(* POU FB_KL3208Config, ST *)
FUNCTION_BLOCK FB_KL3208Config
VAR_INPUT
	bConfigurate		: BOOL; 		(*Rising edge starts configuration including read-configuration afterwards*)
	bReadConfig			: BOOL;			(*Rising edge reads the actual configuration*)
	iSetSensorType		: INT;			(*Sensor-type to be set, see table*)
	tTimeout			: TIME :=t#5s;	(*Time-out-time for Reading/Configuration - initially set to 5s*)
END_VAR
VAR_OUTPUT
	bBusy				: BOOL;			(*Reading or configuration is in progress*)
	bError				: BOOL;			(*Error while reading/configuration*)
	iErrorId			: UDINT;		(*Id of the last upcoming error*)
	iState				: USINT;		(*As long as the funcion-block is not busy, this variable shows the state of the terminal, otherwise it is 0*)
	iDataIn				: INT;			(*As long as the funcion-block is not busy, this variable shows the dataIn of the terminal, otherwise it keeps the value previous to reding/configuration*)
	iTerminalType		: WORD;			(*Terminal-type-number, in this case 3208*)
	iSpecialType		: WORD;			(*Sub-type-number*)
	iFirmwareVersion	: WORD;			(*Firmware in ASCII-code*)
	sDescription		: STRING;		(*Terminal-type, special-type and firmware-version as readable text*)
	sSensorType			: STRING;		(*Text-description of entered sensor-type*)
END_VAR
VAR
	rtRead				: R_TRIG;
	rtSet				: R_TRIG;
	bSetReq				: BOOL;
	tonTimeout			: TON;
	iStep				: INT;
	bSetConfigError		: BOOL;
	wReg32				: WORD;
	wSetReg32			: WORD;
	wReg39				: WORD;
	wSetReg39			: WORD;
	wFirmware			: WORD;
	pFirmware			: POINTER TO WORD;
	sFirmware			: STRING(2);
	iDataInSaved		: INT;
END_VAR
VAR_IN_OUT
	stInData   			: ST_KL3208InData;	(* Process image of the inputs. *)
	stOutData 			: ST_KL3208OutData;	(* Process image of the outputs. *)
END_VAR
tonTimeout	(PT:=tTimeout);
IF	tonTimeout.Q	THEN
	bError			:= TRUE;
	iErrorId		:= 16#8001;
	iStep			:= 0;
END_IF

rtSet	(CLK:=bConfigurate);
rtRead	(CLK:=bReadConfig);

IF	(rtSet.Q OR rtRead.Q)	AND NOT bBusy THEN
	bBusy			:= TRUE;
	bError			:= FALSE;
	iErrorId		:= 0;
	iDataInSaved	:= stInData.iDataIn;
	tonTimeout.IN	:= TRUE;
	iStep			:= 10;
	IF	rtSet.Q	THEN
		bSetReq	:= TRUE;
	END_IF
END_IF

IF bBusy THEN
	iDataIn		:= iDataInSaved;
	iState		:= 0;
ELSE
	iDataIn		:= stInData.iDataIn;
	iState		:= stInData.iState;
END_IF


CASE iStep OF

0:	(*idle*)
	bBusy				:= FALSE;
	bSetReq				:= FALSE;
	tonTimeout.IN		:= FALSE;

10:	(*Klemmentyp (Kl32xx) auslesen: Register 8*)
	stOutData.iCtrl	:= 16#88;	(*Register 8 Lesen*)

	IF stInData.iState = 16#88 THEN
		iTerminalType	:= INT_TO_WORD(stInData.iDataIn);
		iStep:=20;
	END_IF

20:	(*Spezialtyp (Kl32xx-yyy) auslesen: Register 29*)
	stOutData.iCtrl	:= 16#9D;	(*Register 29 Lesen*)

	IF stInData.iState = 16#9D THEN
		iSpecialType	:= INT_TO_WORD(stInData.iDataIn);
		iStep:=30;
	END_IF

30:	(*Firmware auslesen: Register 9*)
	stOutData.iCtrl	:= 16#89;	(*Register 9 Lesen*)

	IF stInData.iState = 16#89 THEN
		iFirmwareVersion:= INT_TO_WORD(stInData.iDataIn);
		(*Umwandlung in STRING*)
		wFirmware		:= iFirmwareVersion;
		wFirmware		:= ROR(wFirmware,8);(*Reihenfolge der beiden Zeichen der Firmware tauschen*)
		pFirmware		:= ADR(sFirmware);	(*Einen Pointer auf den Info-String (Ausgang) legen*)
		pFirmware^		:= wFirmware;		(*Diesen Adressbereich mit dem richtig getauschen Wert beschreiben - damit ist auch der String beschrieben*)

		sDescription	:= CONCAT('Terminal ',WORD_TO_STRING(iTerminalType));

		CASE LEN(WORD_TO_STRING(iSpecialType)) OF
			1: sDescription	:= CONCAT(sDescription,'-000');
			2: sDescription	:= CONCAT(sDescription,'-00');
			3: sDescription	:= CONCAT(sDescription,'-0');
		ELSE
			sDescription	:= CONCAT(sDescription,'-');
		END_CASE

		sDescription	:= CONCAT(sDescription,WORD_TO_STRING(iSpecialType));
		sDescription	:= CONCAT(sDescription,' / Firmware ');
		sDescription	:= CONCAT(sDescription,sFirmware);

		IF bSetReq	THEN
			iStep:=100;
		ELSE
			iStep:=150;
		END_IF
	END_IF

	(*Falscher Klemmentyp angeschlossen, Konfiguration vorzeitig abbrechen*)
	IF (iTerminalType <> 3208)	THEN
		bError		:= TRUE;
		iErrorId	:= 16#8002;
		iStep		:= 160;
	END_IF

(*-----------------------------------------------------------------*)

100:(*jetzige Sensoreinstellung lesen: Register 32*)
	stOutData.iCtrl	:= 16#A0;	(*Register 32 Lesen*)

	IF stInData.iState = 16#A0 THEN
		wReg32			:= INT_TO_WORD(stInData.iDataIn);
		iStep:=105;
	END_IF

105:(*jetzige Sensoreinstellung lesen: Register 39*)
	stOutData.iCtrl	:= 16#A7;	(*Register 39 Lesen*)

	IF stInData.iState = 16#A7 THEN
		wReg39			:= INT_TO_WORD(stInData.iDataIn);
		A_SetConfigTable;			(*entsprechende Einstellungen vornehmen*)
		iStep:=110;
		IF	bSetConfigError	THEN
			iStep:=150;
		END_IF
	END_IF

110:(*Codewort Register 31 setzen: 16#1235 -> Schreibschutz aufheben*)
	stOutData.iCtrl	:= 16#DF;	(*Register 31 beschreiben*)
	stOutData.iDataOut	:= 16#1235;	(*Nutzdaten: Codewort*)

	IF stInData.iState = 16#9F THEN
		stOutData.iCtrl	:= 16#9F;	(*Register 31 Auslesen*)
		iStep:=120;
	END_IF

120:(*Bestätigung Codewort gesetzt erfragen*)
	IF	stInData.iDataIn	= 16#1235	THEN
		iStep:=130;
	END_IF

130:(*Nun Register 32 mit dem neuen Wert beschreiben*)
	stOutData.iCtrl	:= 16#E0;	(*Register 32 beschreiben*)
	stOutData.iDataOut	:= WORD_TO_INT(wSetReg32);

	IF stInData.iState = 16#A0 THEN
		iStep:=135;
	END_IF

135:(*Und Register 39 mit dem neuen Wert beschreiben*)
	stOutData.iCtrl	:= 16#E7;	(*Register 39 beschreiben*)
	stOutData.iDataOut	:= WORD_TO_INT(wSetReg39);

	IF stInData.iState = 16#A7 THEN
		iStep:=140;
	END_IF

140:(*Codewort Register 31 löschen: 16#0000 -> Schreibschutz setzen*)
	stOutData.iCtrl	:= 16#DF;	(*Register 31 beschreiben*)
	stOutData.iDataOut	:= 16#0000;

	IF stInData.iState = 16#9F THEN
		iStep:=150;
	END_IF

150:(*nach erfolgter Parametrierung Sensoreinstellung lesen: Register 32*)
	stOutData.iCtrl	:= 16#A0;	(*Register 32 Lesen*)

	IF stInData.iState = 16#A0 THEN
		wReg32			:= INT_TO_WORD(stInData.iDataIn);
		iStep:=155;
	END_IF

155:(*nach erfolgter Parametrierung Sensoreinstellung lesen: Register 39*)
	stOutData.iCtrl	:= 16#A7;	(*Register 39 Lesen*)

	IF stInData.iState = 16#A7 THEN
		wReg39			:= INT_TO_WORD(stInData.iDataIn);
		A_ReadConfigTable;
		iStep:=160;
	END_IF

160:(*Registerkommunikation beenden*)
	stOutData.iCtrl	:= 0; (*auch alle anderen Steuerbits mit ablöschen*)
	(*Rückmeldeabfrage Prozessdatenaustausch (Bit7) noch aktiv? *)
	(*alle anderen Bits könnten durch einen bestimmten Signalpegel gesetzt sein *)
	IF stInData.iState.7 = FALSE THEN
		iStep:=0;
	END_IF

END_CASE
END_FUNCTION_BLOCK
ACTION A_ReadConfigTable:
(*IF Reg39 is set to 0, Reg32 is responsible for the sensor-type, otherwise Reg39 sets the sensor*)

IF	wReg39=0	THEN
	CASE (SHR(wReg32,12)) OF	(*Check sensor-type via the 4 most significant bits*)
		2#0000: sSensorType	:= 'PT1000';
		2#0001: sSensorType	:= 'NI1000';
		2#0010: sSensorType	:= 'RSNI1000';
	ELSE
		sSensorType	:='Unknown';
		bError		:= TRUE;
		iErrorId	:= 16#8021;
	END_CASE
ELSE
	CASE wReg39 OF
		16#32: sSensorType	:= 'NCT1K8';
		16#33: sSensorType	:= 'NCT1K8_TK';
		16#34: sSensorType	:= 'NCT2K2';
		16#35: sSensorType	:= 'NCT3K';
		16#36: sSensorType	:= 'NCT5K';
		16#37: sSensorType	:= 'NTC10K';
		16#38: sSensorType	:= 'NTC10KPRE';
		16#39: sSensorType	:= 'NTC10K_3204';
		16#3A: sSensorType	:= 'NTC10KTYP2';
		16#3B: sSensorType	:= 'NTC10KTYP3';
		16#3C: sSensorType	:= 'NTC10KDALE';
		16#3D: sSensorType	:= 'NTC10K3A221';
		16#3E: sSensorType	:= 'NTC20K';
		16#64: sSensorType	:= 'Poti, Resolution 0,1 Ohm';
		16#65: sSensorType	:= 'Poti, Resolution 1 Ohm';
		16#C8: sSensorType	:= 'NTC100K';
		16#FF: sSensorType	:= 'User defined';
	ELSE
		sSensorType	:='Unknown';
		bError		:= TRUE;
		iErrorId	:= 16#8021;
	END_CASE
END_IF
END_ACTION
ACTION A_SetConfigTable:
bSetConfigError	:= FALSE;

CASE iSetSensorType OF	(*Then set the sensor-type via the 4 most significant bits*)

	0:	wSetReg32	:= wReg32		AND 2#0000111111111111;(*First clear the first 4 bits*)
		wSetReg32	:= wSetReg32	OR 2#0000000000000000;(*PT1000*)	(*Then set the sensor-type via the 4 most significant bits*)
		wSetReg39	:= 0;

	1:	wSetReg32	:= wReg32		AND 2#0000111111111111;(*First clear the first 4 bits*)
		wSetReg32	:= wSetReg32	OR 2#0001000000000000;(*NI1000*)	(*Then set the sensor-type via the 4 most significant bits*)
		wSetReg39	:= 0;

	2:	wSetReg32	:= wReg32		AND 2#0000111111111111;(*First clear the first 4 bits*)
		wSetReg32	:= wSetReg32	OR 2#0010000000000000;(*RSNI1000*)	(*Then set the sensor-type via the 4 most significant bits*)
		wSetReg39	:= 0;


	3:	wSetReg39	:= 16#32;		(*NCT1K8*)
	4:	wSetReg39	:= 16#33;		(*NCT1K8_TK*)
	5:	wSetReg39	:= 16#34;		(*NCT2K2*)
	6:	wSetReg39	:= 16#35;		(*NCT3K*)
	7:	wSetReg39	:= 16#36;		(*NCT5K*)
	8:	wSetReg39	:= 16#37;		(*NTC10K*)
	9:	wSetReg39	:= 16#38;		(*NTC10KPRE*)
	10:	wSetReg39	:= 16#39;		(*NTC10K_3204*)
	11:	wSetReg39	:= 16#3A;		(*NTC10KTYP2*)
	12:	wSetReg39	:= 16#3B;		(*NTC10KTYP3*)
	13:	wSetReg39	:= 16#3C;		(*NTC10KDALE*)
	14:	wSetReg39	:= 16#3D;		(*NTC10K3A221*)
	15:	wSetReg39	:= 16#3E;		(*NTC20K*)
	16:	wSetReg39	:= 16#64;		(*Poti, Resolution 0,1 Ohm*)
	17:	wSetReg39	:= 16#65;		(*Poti, Resolution 1 Ohm*)
	18:	wSetReg39	:= 16#C8;		(*NTC100K*)
ELSE
	bSetConfigError	:= TRUE;
	bError			:= TRUE;
	iErrorId		:= 16#8020;
END_CASE
END_ACTION

(* POU FB_KL320xConfig, ST *)
FUNCTION_BLOCK FB_KL320xConfig
VAR_INPUT
	bConfigurate		: BOOL; 		(*Rising edge starts configuration including read-configuration afterwards*)
	bReadConfig			: BOOL;			(*Rising edge reads the actual configuration*)
	iSetSensorType		: INT;			(*Sensor-type to be set, see table*)
	tTimeout			: TIME :=t#5s;	(*Time-out-time for Reading/Configuration - initially set to 5s*)
END_VAR
VAR_OUTPUT
	bBusy				: BOOL;			(*Reading or configuration is in progress*)
	bError				: BOOL;			(*Error while reading/configuration*)
	iErrorId			: UDINT;		(*Id of the last upcoming error*)
	iState				: USINT;		(*As long as the funcion-block is not busy, this variable shows the state of the terminal, otherwise it is 0*)
	iDataIn				: INT;			(*As long as the funcion-block is not busy, this variable shows the dataIn of the terminal, otherwise it keeps the value previous to reding/configuration*)
	iTerminalType		: WORD;			(*Terminal-type-number, e.g. 3204*)
	iSpecialType		: WORD;			(*Sub-type-number*)
	iFirmwareVersion	: WORD;			(*Firmware in ASCII-code*)
	sDescription		: STRING;		(*Terminal-type, special-type and firmware-version as readable text*)
	sSensorType			: STRING;		(*Text-description of entered sensor-type*)
	bTwoWiredConnection	: BOOL;			(*Shows, if two-wired connection is selected*)
END_VAR
VAR
	rtRead				: R_TRIG;
	rtSet				: R_TRIG;
	bSetReq				: BOOL;
	tonTimeout			: TON;
	iStep				: INT;
	bSetConfigError		: BOOL;
	wReg32				: WORD;
	wSetReg32			: WORD;
	wFirmware			: WORD;
	pFirmware			: POINTER TO WORD;
	sFirmware			: STRING(2);
	iDataInSaved		: INT;
END_VAR
VAR_IN_OUT
	stInData   			: ST_KL320xInData;	(* Process image of the inputs. *)
	stOutData 			: ST_KL320xOutData;	(* Process image of the outputs. *)
END_VAR
tonTimeout	(PT:=tTimeout);
IF	tonTimeout.Q	THEN
	bError			:= TRUE;
	iErrorId		:= 16#8001;
	iStep			:= 0;
END_IF

rtSet	(CLK:=bConfigurate);
rtRead	(CLK:=bReadConfig);

IF	(rtSet.Q OR rtRead.Q)	AND NOT bBusy THEN
	bBusy			:= TRUE;
	bError			:= FALSE;
	iErrorId		:= 0;
	iDataInSaved	:= stInData.iDataIn;
	tonTimeout.IN	:= TRUE;
	iStep			:= 10;
	IF	rtSet.Q	THEN
		bSetReq	:= TRUE;
	END_IF
END_IF

IF bBusy THEN
	iDataIn		:= iDataInSaved;
	iState		:= 0;
ELSE
	iDataIn		:= stInData.iDataIn;
	iState		:= stInData.iState;
END_IF


CASE iStep OF

0:	(*idle*)
	bBusy				:= FALSE;
	bSetReq				:= FALSE;
	tonTimeout.IN		:= FALSE;

10:	(*Klemmentyp (Kl32xx) auslesen: Register 8*)
	stOutData.iCtrl	:= 16#88;	(*Register 8 Lesen*)

	IF stInData.iState = 16#88 THEN
		iTerminalType	:= INT_TO_WORD(stInData.iDataIn);
		iStep:=20;
	END_IF

20:	(*Spezialtyp (Kl32xx-yyy) auslesen: Register 29*)
	stOutData.iCtrl	:= 16#9D;	(*Register 29 Lesen*)

	IF stInData.iState = 16#9D THEN
		iSpecialType	:= INT_TO_WORD(stInData.iDataIn);
		iStep:=30;
	END_IF

30:	(*Firmware auslesen: Register 9*)
	stOutData.iCtrl	:= 16#89;	(*Register 9 Lesen*)

	IF stInData.iState = 16#89 THEN
		iFirmwareVersion:= INT_TO_WORD(stInData.iDataIn);
		(*Umwandlung in STRING*)
		wFirmware		:= iFirmwareVersion;
		wFirmware		:= ROR(wFirmware,8);(*Reihenfolge der beiden Zeichen der Firmware tauschen*)
		pFirmware		:= ADR(sFirmware);	(*Einen Pointer auf den Info-String (Ausgang) legen*)
		pFirmware^		:= wFirmware;		(*Diesen Adressbereich mit dem richtig getauschen Wert beschreiben - damit ist auch der String beschrieben*)

		sDescription	:= CONCAT('Terminal ',WORD_TO_STRING(iTerminalType));

		CASE LEN(WORD_TO_STRING(iSpecialType)) OF
			1: sDescription	:= CONCAT(sDescription,'-000');
			2: sDescription	:= CONCAT(sDescription,'-00');
			3: sDescription	:= CONCAT(sDescription,'-0');
		ELSE
			sDescription	:= CONCAT(sDescription,'-');
		END_CASE

		sDescription	:= CONCAT(sDescription,WORD_TO_STRING(iSpecialType));
		sDescription	:= CONCAT(sDescription,' / Firmware ');
		sDescription	:= CONCAT(sDescription,sFirmware);

		IF bSetReq	THEN
			iStep:=100;
		ELSE
			iStep:=150;
		END_IF
	END_IF

	(*Falscher Klemmentyp angeschlossen, Konfiguration vorzeitig abbrechen*)
	IF ((iTerminalType <> 3201)	AND (iTerminalType <> 3202) AND (iTerminalType <> 3204))	THEN
		bError		:= TRUE;
		iErrorId	:= 16#8002;
		iStep		:= 160;
	END_IF

(*-----------------------------------------------------------------*)

100:(*jetzige Sensoreinstellung lesen: Register 32*)
	stOutData.iCtrl	:= 16#A0;	(*Register 32 Lesen*)

	IF stInData.iState = 16#A0 THEN
		wReg32			:= INT_TO_WORD(stInData.iDataIn);
		A_SetConfigTable;		(*entsprechende Bits für den zu schreibenden Wert setzen, der Rest bleibt unberührt*)
		iStep:=110;
		IF	bSetConfigError	THEN
			iStep:=150;
		END_IF
	END_IF

110:(*Codewort Register 31 setzen: 16#1235 -> Schreibschutz aufheben*)
	stOutData.iCtrl	:= 16#DF;	(*Register 31 beschreiben*)
	stOutData.iDataOut	:= 16#1235;	(*Nutzdaten: Codewort*)

	IF stInData.iState = 16#9F THEN
		stOutData.iCtrl	:= 16#9F;	(*Register 31 Auslesen*)
		iStep:=120;
	END_IF

120:(*Bestätigung Codewort gesetzt erfragen*)
	IF	stInData.iDataIn	= 16#1235	THEN
		iStep:=130;
	END_IF

130:(*Nun Register 32 mit dem neuen Wert beschreiben*)
	stOutData.iCtrl	:= 16#E0;	(*Register 32 beschreiben*)
	stOutData.iDataOut	:= WORD_TO_INT(wSetReg32);

	IF stInData.iState = 16#A0 THEN
		iStep:=140;
	END_IF

140:(*Codewort Register 31 löschen: 16#0000 -> Schreibschutz setzen*)
	stOutData.iCtrl	:= 16#DF;	(*Register 31 beschreiben*)
	stOutData.iDataOut	:= 16#0000;

	IF stInData.iState = 16#9F THEN
		iStep:=150;
	END_IF

150:(*nach erfolgter Parametrierung Sensoreinstellung lesen: Register 32*)
	stOutData.iCtrl	:= 16#A0;	(*Register 32 Lesen*)

	IF stInData.iState = 16#A0 THEN
		wReg32			:= INT_TO_WORD(stInData.iDataIn);
		A_ReadConfigTable;
		iStep:=160;
	END_IF

160:(*Registerkommunikation beenden*)
	stOutData.iCtrl	:= 0; (*auch alle anderen Steuerbits mit ablöschen*)
	(*Rückmeldeabfrage Prozessdatenaustausch (Bit7) noch aktiv? *)
	(*alle anderen Bits könnten durch einen bestimmten Signalpegel gesetzt sein *)
	IF stInData.iState.7 = FALSE THEN
		iStep:=0;
	END_IF

END_CASE
END_FUNCTION_BLOCK
ACTION A_ReadConfigTable:
CASE (SHR(wReg32,12)) OF	(*Check sensor-type via the 4 most significant bits*)
	2#0000: sSensorType:='PT100';
	2#0001: sSensorType:='NI100';
	2#0010: sSensorType:='PT1000';
	2#0011: sSensorType:='PT500';
	2#0100: sSensorType:='PT200';
	2#0101: sSensorType:='NI1000';
	2#0110: sSensorType:='NI120';
	
	2#1110: sSensorType:='10Ohm .. 5000Ohm';
	2#1111: sSensorType:='10Ohm .. 1200Ohm';
ELSE
	sSensorType	:='Unknown';
	bError		:= TRUE;
	iErrorId	:= 16#802A;
END_CASE

bTwoWiredConnection:=wReg32.10;
END_ACTION
ACTION A_SetConfigTable:
bSetConfigError	:= FALSE;

wSetReg32:=wReg32 AND 2#0000111111111111;(*First clear the first 4 bits*)

CASE iSetSensorType OF	(*Then set the sensor-type via the 4 most significant bits - Bit 10 sets 2-wired-connection*)

	0:	wSetReg32:=wSetReg32 OR 2#0000000000000000;(*PT100*)
		wSetReg32.10:=FALSE;					(*1-Wired*)

	1:	wSetReg32:=wSetReg32 OR 2#0001000000000000;(*NI100*)
		wSetReg32.10:=FALSE;					(*1-Wired*)

	2:	wSetReg32:=wSetReg32 OR 2#0010000000000000;(*PT1000*)
		wSetReg32.10:=FALSE;					(*1-Wired*)

	3:	wSetReg32:=wSetReg32 OR 2#0011000000000000;(*PT500*)
		wSetReg32.10:=FALSE;					(*1-Wired*)

	4:	wSetReg32:=wSetReg32 OR 2#0100000000000000;(*PT200*)
		wSetReg32.10:=FALSE;					(*1-Wired*)

	5:	wSetReg32:=wSetReg32 OR 2#0101000000000000;(*NI1000*)
		wSetReg32.10:=FALSE;					(*1-Wired*)

	6:	wSetReg32:=wSetReg32 OR 2#0110000000000000;(*NI120*)
		wSetReg32.10:=FALSE;					(*1-Wired*)

	7:	wSetReg32:=wSetReg32 OR 2#1110000000000000;(*10Ohm .. 5000Ohm*)
		wSetReg32.10:=FALSE;					(*1-Wired*)

	8:	wSetReg32:=wSetReg32 OR 2#1111000000000000;(*10Ohm .. 1200Ohm*)
		wSetReg32.10:=FALSE;					(*1-Wired*)

	9:	wSetReg32:=wSetReg32 OR 2#0010000000000000;(*PT1000*)
		wSetReg32.10:=TRUE;						(*2-Wired*)

		IF (iTerminalType=3204)	THEN			(*2-Wired is not allowed for KL3204*)
			bSetConfigError	:= TRUE;
			bError			:= TRUE;
			iErrorId		:= 16#8028;
		END_IF
ELSE
	bSetConfigError	:= TRUE;
	bError			:= TRUE;
	iErrorId		:= 16#8029;
END_CASE
END_ACTION

(* POU FB_KL3228Config, ST *)
FUNCTION_BLOCK FB_KL3228Config
VAR_INPUT
	bConfigurate		: BOOL; 		(*Rising edge starts configuration including read-configuration afterwards*)
	bReadConfig			: BOOL;			(*Rising edge reads the actual configuration*)
	iSetSensorType		: INT;			(*Sensor-type to be set, see table*)
	tTimeout			: TIME :=t#5s;	(*Time-out-time for Reading/Configuration - initially set to 5s*)
END_VAR
VAR_OUTPUT
	bBusy				: BOOL;			(*Reading or configuration is in progress*)
	bError				: BOOL;			(*Error while reading/configuration*)
	iErrorId			: UDINT;		(*Id of the last upcoming error*)
	iState				: USINT;		(*As long as the funcion-block is not busy, this variable shows the state of the terminal, otherwise it is 0*)
	iDataIn				: INT;			(*As long as the funcion-block is not busy, this variable shows the dataIn of the terminal, otherwise it keeps the value previous to reding/configuration*)
	iTerminalType		: WORD;			(*Terminal-type-number, in this case 3228*)
	iSpecialType		: WORD;			(*Sub-type-number*)
	iFirmwareVersion	: WORD;			(*Firmware in ASCII-code*)
	sDescription		: STRING;		(*Terminal-type, special-type and firmware-version as readable text*)
	sSensorType			: STRING;		(*Text-description of entered sensor-type*)
END_VAR
VAR
	rtRead				: R_TRIG;
	rtSet				: R_TRIG;
	bSetReq				: BOOL;
	tonTimeout			: TON;
	iStep				: INT;
	bSetConfigError		: BOOL;
	wReg32				: WORD;
	wSetReg32			: WORD;
	wFirmware			: WORD;
	pFirmware			: POINTER TO WORD;
	sFirmware			: STRING(2);
	iDataInSaved		: INT;
END_VAR
VAR_IN_OUT
	stInData   			: ST_KL3228InData;	(* Process image of the inputs. *)
	stOutData 			: ST_KL3228OutData;	(* Process image of the outputs. *)
END_VAR
tonTimeout	(PT:=tTimeout);
IF	tonTimeout.Q	THEN
	bError			:= TRUE;
	iErrorId		:= 16#8001;
	iStep			:= 0;
END_IF

rtSet	(CLK:=bConfigurate);
rtRead	(CLK:=bReadConfig);

IF	(rtSet.Q OR rtRead.Q)	AND NOT bBusy THEN
	bBusy			:= TRUE;
	bError			:= FALSE;
	iErrorId		:= 0;
	iDataInSaved	:= stInData.iDataIn;
	tonTimeout.IN	:= TRUE;
	iStep			:= 10;
	IF	rtSet.Q	THEN
		bSetReq	:= TRUE;
	END_IF
END_IF

IF bBusy THEN
	iDataIn		:= iDataInSaved;
	iState		:= 0;
ELSE
	iDataIn		:= stInData.iDataIn;
	iState		:= stInData.iState;
END_IF


CASE iStep OF

0:	(*idle*)
	bBusy				:= FALSE;
	bSetReq				:= FALSE;
	tonTimeout.IN		:= FALSE;

10:	(*Klemmentyp (Kl32xx) auslesen: Register 8*)
	stOutData.iCtrl	:= 16#88;	(*Register 8 Lesen*)

	IF stInData.iState = 16#88 THEN
		iTerminalType	:= INT_TO_WORD(stInData.iDataIn);
		iStep:=20;
	END_IF

20:	(*Spezialtyp (Kl32xx-yyy) auslesen: Register 29*)
	stOutData.iCtrl	:= 16#9D;	(*Register 29 Lesen*)

	IF stInData.iState = 16#9D THEN
		iSpecialType	:= INT_TO_WORD(stInData.iDataIn);
		iStep:=30;
	END_IF

30:	(*Firmware auslesen: Register 9*)
	stOutData.iCtrl	:= 16#89;	(*Register 9 Lesen*)

	IF stInData.iState = 16#89 THEN
		iFirmwareVersion:= INT_TO_WORD(stInData.iDataIn);
		(*Umwandlung in STRING*)
		wFirmware		:= iFirmwareVersion;
		wFirmware		:= ROR(wFirmware,8);(*Reihenfolge der beiden Zeichen der Firmware tauschen*)
		pFirmware		:= ADR(sFirmware);	(*Einen Pointer auf den Info-String (Ausgang) legen*)
		pFirmware^		:= wFirmware;		(*Diesen Adressbereich mit dem richtig getauschen Wert beschreiben - damit ist auch der String beschrieben*)

		sDescription	:= CONCAT('Terminal ',WORD_TO_STRING(iTerminalType));

		CASE LEN(WORD_TO_STRING(iSpecialType)) OF
			1: sDescription	:= CONCAT(sDescription,'-000');
			2: sDescription	:= CONCAT(sDescription,'-00');
			3: sDescription	:= CONCAT(sDescription,'-0');
		ELSE
			sDescription	:= CONCAT(sDescription,'-');
		END_CASE

		sDescription	:= CONCAT(sDescription,WORD_TO_STRING(iSpecialType));
		sDescription	:= CONCAT(sDescription,' / Firmware ');
		sDescription	:= CONCAT(sDescription,sFirmware);

		IF bSetReq	THEN
			iStep:=100;
		ELSE
			iStep:=150;
		END_IF
	END_IF

	(*Falscher Klemmentyp angeschlossen, Konfiguration vorzeitig abbrechen*)
	IF (iTerminalType <> 3228)	THEN
		bError		:= TRUE;
		iErrorId	:= 16#8002;
		iStep		:= 160;
	END_IF

(*-----------------------------------------------------------------*)

100:(*jetzige Sensoreinstellung lesen: Register 32*)
	stOutData.iCtrl	:= 16#A0;	(*Register 32 Lesen*)

	IF stInData.iState = 16#A0 THEN
		wReg32			:= INT_TO_WORD(stInData.iDataIn);
		A_SetConfigTable;		(*entsprechende Bits für den zu schreibenden Wert setzen, der Rest bleibt unberührt*)
		iStep:=110;
		IF	bSetConfigError	THEN
			iStep:=150;
		END_IF
	END_IF

110:(*Codewort Register 31 setzen: 16#1235 -> Schreibschutz aufheben*)
	stOutData.iCtrl	:= 16#DF;	(*Register 31 beschreiben*)
	stOutData.iDataOut	:= 16#1235;	(*Nutzdaten: Codewort*)

	IF stInData.iState = 16#9F THEN
		stOutData.iCtrl	:= 16#9F;	(*Register 31 Auslesen*)
		iStep:=120;
	END_IF

120:(*Bestätigung Codewort gesetzt erfragen*)
	IF	stInData.iDataIn	= 16#1235	THEN
		iStep:=130;
	END_IF

130:(*Nun Register 32 mit dem neuen Wert beschreiben*)
	stOutData.iCtrl	:= 16#E0;	(*Register 32 beschreiben*)
	stOutData.iDataOut	:= WORD_TO_INT(wSetReg32);

	IF stInData.iState = 16#A0 THEN
		iStep:=140;
	END_IF

140:(*Codewort Register 31 löschen: 16#0000 -> Schreibschutz setzen*)
	stOutData.iCtrl	:= 16#DF;	(*Register 31 beschreiben*)
	stOutData.iDataOut	:= 16#0000;

	IF stInData.iState = 16#9F THEN
		iStep:=150;
	END_IF

150:(*nach erfolgter Parametrierung Sensoreinstellung lesen: Register 32*)
	stOutData.iCtrl	:= 16#A0;	(*Register 32 Lesen*)

	IF stInData.iState = 16#A0 THEN
		wReg32			:= INT_TO_WORD(stInData.iDataIn);
		A_ReadConfigTable;
		iStep:=160;
	END_IF

160:(*Registerkommunikation beenden*)
	stOutData.iCtrl	:= 0; (*auch alle anderen Steuerbits mit ablöschen*)
	(*Rückmeldeabfrage Prozessdatenaustausch (Bit7) noch aktiv? *)
	(*alle anderen Bits könnten durch einen bestimmten Signalpegel gesetzt sein *)
	IF stInData.iState.7 = FALSE THEN
		iStep:=0;
	END_IF

END_CASE
END_FUNCTION_BLOCK
ACTION A_ReadConfigTable:
CASE (SHR(wReg32,12)) OF	(*Check sensor-type via the 4 most significant bits*)
	2#0000: sSensorType	:= 'PT1000';
	2#0001: sSensorType	:= 'NI1000';
	2#0010: sSensorType	:= 'RSNI1000';
ELSE
	sSensorType	:='Unknown';
	bError		:= TRUE;
	iErrorId	:= 16#8031;
END_CASE
END_ACTION
ACTION A_SetConfigTable:
bSetConfigError	:= FALSE;

CASE iSetSensorType OF	(*Then set the sensor-type via the 4 most significant bits*)
	0:	wSetReg32	:= wReg32		AND 2#0000111111111111;(*First clear the first 4 bits*)
		wSetReg32	:= wSetReg32	OR 2#0000000000000000;(*PT1000*)	(*Then set the sensor-type via the 4 most significant bits*)

	1:	wSetReg32	:= wReg32		AND 2#0000111111111111;(*First clear the first 4 bits*)
		wSetReg32	:= wSetReg32	OR 2#0001000000000000;(*NI1000*)	(*Then set the sensor-type via the 4 most significant bits*)

	2:	wSetReg32	:= wReg32		AND 2#0000111111111111;(*First clear the first 4 bits*)
		wSetReg32	:= wSetReg32	OR 2#0010000000000000;(*RSNI1000*)(*Then set the sensor-type via the 4 most significant bits*)
ELSE
	bSetConfigError	:= TRUE;
	bError			:= TRUE;
	iErrorId		:= 16#8030;
END_CASE
END_ACTION

(* POU FB_NovRamReadWrite, ST *)
FUNCTION_BLOCK FB_NovRamReadWrite (*if the dpram must be accessed in a special manor, this function block returns error 0x701. In this case use FB_NovRamReadWriteEx instead.*)
VAR_INPUT
	nDevId 	: UDINT;		(* Device id of the FCxxxx card. Map the FC card as generic DPRAM/NOVRAM card im System Manager *)
	bRead		: BOOL;		(* Rising edge starts read data block from NovRam*)
	bWrite		: BOOL;		(* Rising edge starts write data block to NovRam*)
	cbSrcLen	: UDINT;		(* Number of data bytes to write *)
	cbDestLen: UDINT;		(* Number of data bytes to read*)
	pSrcAddr	: UDINT;		(* Address of the write data buffer *)
	pDestAddr	: UDINT;		(* Address of the read data buffer *)
	tTimeOut	: TIME := DEFAULT_ADS_TIMEOUT;		(* Max timeout for this command *)
END_VAR
VAR_OUTPUT
	bBusy		: BOOL;		(* The fb is working *)
	bError		: BOOL;		(* The fb returns an error *)
	nErrId		: UDINT;		(* Error code *)
	cbRead	: UDINT;		(* Number of succesfully read data bytes *)
	cbWrite	: UDINT;		(* Number of succesfully write data bytes *)
END_VAR
VAR
	bInit			: BOOL := FALSE;
	nInitDevId		: UDINT	:= 0;
	bWantRead		: BOOL := FALSE;
	bWantWrite		: BOOL := FALSE;

	iStep			: BYTE := 0;
	RisingRead		: R_TRIG;
	RisingWrite		: R_TRIG;
	stNovRamAddrInfo: ST_NovRamAddrInfo;
	fbAdsReadEx		: ADSREADEX;
END_VAR
RisingRead( CLK := bRead );
RisingWrite( CLK := bWrite );

CASE iStep OF
0:
	(* idle step, wait for rising edge on fb input*)
	IF RisingRead.Q OR RisingWrite.Q THEN

		bBusy 	:= TRUE;
		bError 	:= FALSE;
		nErrId 	:= 0;
		cbRead 	:= 0;
		cbWrite := 0;

		bWantRead 	:=	RisingRead.Q;	(* Save flags *)
		bWantWrite 	:= 	RisingWrite.Q;

		IF	 (nDevId > 0) AND (pSrcAddr > 0) AND (cbSrcLen > 0) AND (pDestAddr > 0) AND (cbDestLen> 0) THEN

			IF 	( NOT bInit ) OR ( bInit AND ( nDevId <> nInitDevId)) THEN

				bInit := FALSE;

				nInitDevId	:= 	nDevId;	(* Save the devid *)
				MEMSET( ADR( stNovRamAddrInfo ) , 0, SIZEOF(stNovRamAddrInfo));

				(* Get the nov ram address pointer and the novram byte size *)
				fbAdsReadEx( READ := FALSE );(*reset the fb*)
				fbAdsReadEx(
						NETID:= '',
						PORT:= AMSPORT_R0_IO,
						IDXGRP:= 16#5000+nInitDevId,
						IDXOFFS:= 16#FFFF_0200,
						LEN:= SIZEOF(stNovRamAddrInfo),
						DESTADDR:= ADR(stNovRamAddrInfo),
						READ:= TRUE,
						TMOUT:= tTimeout);

				iStep := 10;	(* wait for the ads fb *)

			ELSIF bInit THEN

				IF bWantWrite THEN(* copy size bytes to novRAM *)
					cbWrite := MEMCPY(stNovRamAddrInfo.pCardAddress, pSrcAddr, MIN(cbSrcLen,stNovRamAddrInfo.iCardMemSize ) );
				END_IF
				IF bWantRead THEN(* copy size bytes from novRAM *)
					cbRead := MEMCPY(pDestAddr, stNovRamAddrInfo.pCardAddress, MIN(cbDestLen,stNovRamAddrInfo.iCardMemSize ));
				END_IF

				bBusy := FALSE;

			END_IF

		ELSE
			bBusy := FALSE;
			bError := TRUE;
			nErrId := 1798;(* invalid parameter value(s)*)
		END_IF
	END_IF

10:
	fbAdsReadEx( READ := FALSE );
	IF NOT fbAdsReadEx.BUSY THEN

		IF NOT fbAdsReadEx.ERR THEN
			bInit := TRUE;
			bError := FALSE;
			nErrId := 0;

			IF bWantWrite THEN(* copy size bytes to novRAM *)
				cbWrite := MEMCPY(stNovRamAddrInfo.pCardAddress, pSrcAddr, MIN(cbSrcLen,stNovRamAddrInfo.iCardMemSize ) );
			END_IF
			IF bWantRead THEN(* copy size bytes from novRAM *)
				cbRead := MEMCPY(pDestAddr, stNovRamAddrInfo.pCardAddress, MIN(cbDestLen,stNovRamAddrInfo.iCardMemSize ));
			END_IF
		ELSE
			bError := fbAdsReadEx.ERR;
			nErrId := fbAdsReadEx.ERRID;
		END_IF

		bBusy := FALSE;
		iStep := 0; (*go to the idle step and wait for the next call *)

	END_IF

END_CASE;
END_FUNCTION_BLOCK

(* POU FB_NovRamReadWriteEx, ST *)
FUNCTION_BLOCK FB_NovRamReadWriteEx (*if the dpram must be accessed in a special manor, this function block returns error 0x701. In this case use FB_NovRamReadWriteEx instead.*)
VAR_INPUT
	nDevId 		:	UDINT;		(* Device id of the FCxxxx card. Map the FC card as generic DPRAM/NOVRAM card im System Manager *)
	bRead		:	BOOL;		(* Rising edge starts read data block from NovRam*)
	bWrite		:	BOOL;		(* Rising edge starts write data block to NovRam*)
	cbSrcLen	:	UDINT;		(* Number of data bytes to write *)
	cbDestLen	:	UDINT;		(* Number of data bytes to read*)
	pSrcAddr	:	UDINT;		(* Address of the write data buffer *)
	pDestAddr	:	UDINT;		(* Address of the read data buffer *)
	nReadOffs	:	UDINT;		(* Offset in the DPRAM to start reading from*)
	nWriteOffs	:	UDINT;		(* Offset in the DPRAM to start writing to*)
	tTimeOut	: 	TIME;		(* Max timeout for this command *)
END_VAR
VAR_OUTPUT
	bBusy		:	BOOL;		(* The fb is working *)
	bError		:	BOOL;		(* The fb returns an error *)
	nErrId		:	UDINT;		(* Error code *)
	cbRead		: 	UDINT;		(* Number of succesfully read data bytes *)
	cbWrite		: 	UDINT;		(* Number of succesfully write data bytes *)
END_VAR
VAR
	bInit				: BOOL := FALSE;
	nInitDevId		: UDINT	:= 0;
	bWantRead		: BOOL := FALSE;
	bWantWrite		: BOOL := FALSE;
	bCopy			: BOOL := FALSE;

	i				: UDINT:=0;
	iStep			: BYTE := 0;
	RisingRead		: R_TRIG;
	RisingWrite		: R_TRIG;

	stNovRamAddrInfo	: ST_NovRamAddrInfoEx;
	fbAdsReadEx		: ADSREADEX;

	pByte			: POINTER TO BYTE;
	pCard			: POINTER TO BYTE;
END_VAR
RisingRead( CLK := bRead );
RisingWrite( CLK := bWrite );

CASE iStep OF
0:
	(* idle step, wait for rising edge on fb input*)
	IF RisingRead.Q OR RisingWrite.Q THEN

		bBusy 	:= TRUE;
		bError 	:= FALSE;
		nErrId 	:= 0;
		cbRead 	:= 0;
		cbWrite := 0;

		bWantRead 	:=	RisingRead.Q;	(* Save flags *)
		bWantWrite 	:= 	RisingWrite.Q;

		IF	(nDevId > 0) AND (  ( bWantWrite AND ( pSrcAddr>0) AND (cbSrcLen>0) ) OR ( bWantRead AND (pDestAddr > 0) AND (cbDestLen> 0) )  ) THEN
			IF 	( NOT bInit ) OR ( bInit AND ( nDevId <> nInitDevId)) THEN
				bInit := FALSE;

				nInitDevId	:= 	nDevId;	(* Save the devid *)
				MEMSET( ADR( stNovRamAddrInfo ), 0, 10);

				(* Get the nov ram address pointer and the novram byte size *)
				fbAdsReadEx( READ := FALSE );(*reset the fb*)
				fbAdsReadEx(
						NETID:= '',
						PORT:= AMSPORT_R0_IO,
						IDXGRP:= 16#5000+nInitDevId,
						IDXOFFS:= 16#FFFF_0201,
						LEN:= 10,
						DESTADDR:= ADR(stNovRamAddrInfo),
						READ:= TRUE,
						TMOUT:= tTimeout);

				iStep := 10;	(* wait for the ads fb *)

			ELSIF bInit THEN
				bCopy := TRUE;
				bBusy := FALSE;
			END_IF
		ELSE
			bBusy := FALSE;
			bError := TRUE;
			nErrId := 1798;(* invalid parameter value(s)*)
		END_IF
	END_IF

10:
	fbAdsReadEx( READ := FALSE );
	IF NOT fbAdsReadEx.BUSY THEN
		IF NOT fbAdsReadEx.ERR THEN
			bCopy := TRUE;
		ELSE
			bError := fbAdsReadEx.ERR;
			nErrId := fbAdsReadEx.ERRID;
			bBusy := FALSE;
		END_IF
		iStep := 0; (*go to the idle step and wait for the next call *)
	END_IF

END_CASE;

IF bCopy THEN
	IF  (bWantWrite AND (nWriteOffs <= stNovRamAddrInfo.iCardMemSize-1)) OR (bWantRead AND (nReadOffs <= stNovRamAddrInfo.iCardMemSize-1)) THEN
		CASE stNovRamAddrInfo.eAccessType OF
		eIOAccess_Default:
			IF bWantWrite THEN(* copy size bytes to novRAM *)
				cbWrite := MEMCPY(stNovRamAddrInfo.pCardAddress+nWriteOffs, pSrcAddr, MIN(cbSrcLen,stNovRamAddrInfo.iCardMemSize-nWriteOffs) );
			END_IF
			IF bWantRead THEN(* copy size bytes from novRAM *)
				cbRead := MEMCPY(pDestAddr, stNovRamAddrInfo.pCardAddress+nReadOffs, MIN(cbDestLen,stNovRamAddrInfo.iCardMemSize-nReadOffs));
			END_IF
		eIOAccess_Byte:
			IF bWantWrite THEN(* copy size bytes to novRAM *)
				cbWrite:=MIN(cbSrcLen,stNovRamAddrInfo.iCardMemSize-nWriteOffs);
				pByte := pSrcAddr;
				pCard := stNovRamAddrInfo.pCardAddress + nWriteOffs;
				FOR i:=1 TO cbWrite DO
					pCard^:= pByte^;
					pCard := pCard + 1;
					pByte := pByte + 1;
				END_FOR
			END_IF
			IF bWantRead THEN(* copy size bytes from novRAM *)
				cbRead:=MIN(cbDestLen,stNovRamAddrInfo.iCardMemSize-nReadOffs);
				pByte := pDestAddr;
				pCard := stNovRamAddrInfo.pCardAddress + nReadOffs;
				FOR i:=1 TO cbRead  DO
					pByte^:=pCard^;
					pCard := pCard + 1;
					pByte := pByte + 1;
				END_FOR
			END_IF
			bInit := TRUE;
			bError := FALSE;
			nErrId := 0;
		ELSE
			bInit := FALSE;
			bError := TRUE;
			nErrId := 16#701;
		END_CASE
	ELSE
		bInit := FALSE;
		bError := TRUE;
		nErrId := 16#706;
	END_IF
	bBusy := FALSE;
	bCopy:= FALSE;
END_IF
END_FUNCTION_BLOCK

(* POU FB_ReadAdsTecSysData, ST *)
FUNCTION_BLOCK FB_ReadAdsTecSysData
VAR_INPUT
	sNetId		: T_AmsNetId;
	bEnable		: BOOL;
	tCycleTime	: TIME := T#100ms;
END_VAR
VAR_OUTPUT
	bValid		: BOOL;
	bError		: BOOL;
	nErrId		: UDINT;
	stSysData	: ST_AdsTecSysData;
END_VAR
VAR
	dwTemp		: DWORD := 0;
	ptr			: POINTER TO ARRAY[0..3] OF SINT;
	delay		: TON;
	wPort		: WORD := 16#240;
	risingEdge	: R_TRIG;
	step 		: INT := 0;
	fbAdsRdWrtEx: ADSRDWRTEX;
END_VAR
risingEdge( CLK := bEnable );
IF risingEdge.Q THEN
	MEMSET( ADR( stSysData ), 0, SIZEOF( stSysData ) );
	delay( IN := FALSE, PT := tCycleTime );
	bValid := FALSE;
	bError := FALSE;
	nErrId := 0;
	step := 1;
ELSIF (NOT bEnable) THEN
	step := 0;
	bValid := FALSE;
END_IF

CASE step OF
	0:	; (* idle step *)

	1:	(* Wait some time and repeat reading...*)
		delay( IN := TRUE );
		IF delay.Q THEN
			fbAdsRdWrtEx(  WRTRD := FALSE );
			delay( IN := FALSE );
			step := step +1;
		END_IF
	2:
(*	AMSPORT_ROUTER						: UINT := 16#0001;
	ROUTERADSGRP_ACCESS_HARDWARE	: DWORD := 16#0005;
	ROUTERADSOFFS_A_HW_READIOPORT	: DWORD := 16#0001;
*)
		fbAdsRdWrtEx(  WRTRD := FALSE );
		fbAdsRdWrtEx( 	NetId := sNetId,
						Port := 1,
						IDXGRP := 16#05,
						IDXOFFS := 16#01,
						WRITELEN := SIZEOF(wPort),
						READLEN := SIZEOF(dwTemp),
						SRCADDR := ADR( wPort ),
						DESTADDR := ADR( dwTemp ),
						WRTRD := TRUE,
						TMOUT := tCycleTime
						);

		step := step +1;
	3:
		fbAdsRdWrtEx(  WRTRD := FALSE );
		IF NOT fbAdsRdWrtEx.BUSY THEN
			IF NOT fbAdsRdWrtEx.ERR THEN
				stSysData.bShiftKey := GETBIT32( dwTemp, 0 );
				stSysData.bRMouseKey := GETBIT32( dwTemp, 1 );
				stSysData.bHotkey := GETBIT32( dwTemp, 2 );
				stSysData.bTaskChaKey := GETBIT32( dwTemp, 3 );
				stSysData.bABCKey := GETBIT32( dwTemp, 4 );
				stSysData.bRsrv1 := GETBIT32( dwTemp, 5 );
				stSysData.bRsrv2 := GETBIT32( dwTemp,6 );
				stSysData.bRsrv3 := GETBIT32( dwTemp, 7 );

				stSysData.bMainFanErr := GETBIT32( dwTemp, 8 );
				stSysData.bCPUFanErr := GETBIT32( dwTemp, 9 );
				stSysData.bTempErr := GETBIT32( dwTemp, 10 );
				stSysData.bBatteryErr := GETBIT32( dwTemp, 11 );
				stSysData.bRsrv4 := GETBIT32( dwTemp, 12 );
				stSysData.bRsrv5 := GETBIT32( dwTemp, 13 );
				stSysData.bRsrv6 := GETBIT32( dwTemp, 14 );
				stSysData.bRsrv7 := GETBIT32( dwTemp, 15 );

				ptr := ADR( dwTemp );
				stSysData.nMainNTCTemp := ptr^[ 2 ];
				stSysData.nExtNTCTemp := ptr^[ 3 ];
				bValid := TRUE;
				step := 1;
			ELSE
				bValid := FALSE;
				bError := TRUE;
				nErrid := fbAdsRdWrtEx.ERRID;
				step := 0;
			END_IF
		END_IF

			;
END_CASE
END_FUNCTION_BLOCK

(* POU FB_ReadInput_analog, ST *)
(*********************************************************************************************************

NAME..............	:	FB_ReadInput_analog
DATE...............	:	11.07.2003
AUTHOR........	:	G.Sieder (Beckhoff Industrieelektronik)

DESCRIPTION:	FB for Read analog data from one Slave

HISTORY:	
11.07.2003	gs	start coding

*********************************************************************************************************)
FUNCTION_BLOCK FB_ReadInput_analog
VAR_INPUT
	iSlaveaddress		:BYTE;
	iChannel				:BYTE;
	bCycleMode			:BOOL;		(*0: Acyclic , 1:Cyclic (permanent Read/Write) *)
	bStart				:BOOL;
END_VAR
VAR_OUTPUT
	bBusy				:BOOL;
	bErr					:BOOL;
	iErrornumber			:BYTE;
	bValid				:BOOL;
	bOverflow			:BOOL;
	iReadValue			:WORD;

END_VAR
VAR_IN_OUT
	stParameterBuffer		:ST_ParameterBuffer;
END_VAR
VAR
	fbParameterinterface	:FB_ASI_Parameterinterface;
	bHiWord				:BOOL;
	iParametervalue		:DWORD;
	iParameterReadValue	:DWORD;
	iParametergroup		:WORD;
	iErrCounter			:BYTE;
	istate				:INT;
END_VAR
	CASE istate OF

		0:	IF bstart THEN
				bBusy		:=TRUE;
				bErr			:=FALSE;
				bOverflow	:=FALSE;
				bValid		:=FALSE;
				iErrornumber	:=0;
				(*check Slavenumber*)
				IF (iSlaveaddress>64) OR (iChannel>4) THEN
					bErr			:=TRUE;
					iErrornumber	:=ERROR_ASI_SLAVEADDRESS;
					istate		:=10;
				ELSE
					istate		:=1;
				END_IF
			END_IF

		(*prepare Parameternumber*)
		1:	iParametergroup	:=(iSlaveaddress*4)+(iChannel-1);
			istate	:=2;

		(*write Readrequest*)
		2:	fbParameterinterface(iParameternumber	:=iParametergroup+16#200,
							stParameterBuffer		:=stParameterBuffer,
							bParametermode		:=FALSE,
							bCycleMode			:=bCycleMode,
							bStart				:=TRUE);
			IF (NOT fbParameterinterface.bBusy) OR bCycleMode THEN
				IF fbParameterinterface.bErr THEN
					bErr			:=TRUE;
					IF fbParameterinterface.iErrornumber =1 THEN
						iErrornumber	:=ERROR_ASI_COMM_ERROR;
					ELSE
						FOR iErrCounter:=1 TO 3 DO
							IF ((SHR(fbParameterinterface.iErrornumber,iErrCounter-1)) AND 16#2000)<>0 THEN
								iErrornumber :=iErrCounter+10;
							END_IF
						END_FOR
					END_IF
					istate	:=10;
				ELSE
					IF (fbParameterinterface.iParameterReadvalue  AND 16#0200)<>0 THEN
						bOverflow	:=TRUE;
					ELSE
						bValid		:=TRUE;
					END_IF
					iParameterReadValue	:=fbParameterinterface.iParameterReadvalue;
					istate	:=3;
				END_IF
			END_IF

		(*read Parametervalue*)
		3:	iReadValue	:=DWORD_TO_WORD(iParameterReadValue);
			IF (NOT bStart) OR (NOT bCycleMode) THEN
				fbParameterinterface(bStart			:=FALSE,
								stParameterBuffer	:=stParameterBuffer);
				IF (NOT fbParameterinterface.bBusy) THEN
					istate	:=10;
				END_IF
			ELSE
				istate	:=1;
			END_IF

			(*Quit*)
		10:	bBusy	:=FALSE;
			IF (NOT bStart) THEN
				istate	:=0;
			END_IF

	ELSE
		;
	END_CASE
END_FUNCTION_BLOCK

(* POU FB_WriteOutput_analog, ST *)
(*********************************************************************************************************

NAME..............	:	FB_WriteOutput_analog
DATE...............	:	11.07.2003
AUTHOR........	:	G.Sieder (Beckhoff Industrieelektronik)

DESCRIPTION:	FB for Write analog data to one Slave

HISTORY:	
11.07.2003	gs	start coding

*********************************************************************************************************)
FUNCTION_BLOCK FB_WriteOutput_analog
VAR_INPUT
	iSlaveaddress		:BYTE;
	iChannel				:BYTE;
	iSlavevalue			:WORD;
	bCycleMode			:BOOL;		(*0: Acyclic , 1:Cyclic (permanent Read/Write) *)
	bStart				:BOOL;
END_VAR
VAR_OUTPUT
	bBusy				:BOOL;
	bErr					:BOOL;
	iErrornumber			:BYTE;

END_VAR
VAR_IN_OUT
	stParameterBuffer		:ST_ParameterBuffer;
END_VAR
VAR
	fbParameterinterface	:FB_ASI_Parameterinterface;
	bHiWord				:BOOL;
	iParametervalue		:DWORD;
	iParameterReadValue	:DWORD;
	iParametergroup		:WORD;
	iErrCounter			:BYTE;
	istate				:INT;

	iReadValue			:WORD;
END_VAR
	CASE istate OF

		0:	IF bstart THEN
				bBusy		:=TRUE;
				bErr			:=FALSE;
				iErrornumber	:=0;
				(*check Slavenumber*)
				IF (iSlaveaddress>64) OR (iChannel>4) THEN
					bErr			:=TRUE;
					iErrornumber	:=ERROR_ASI_SLAVEADDRESS;
					istate		:=10;
				ELSE
					istate		:=1;
				END_IF
			END_IF

		(*prepare Parameternumber and -value*)
		1:	iParametergroup	:=(iSlaveaddress*4)+(iChannel-1);
			iParametervalue	:=0;
			iParametervalue	:=iSlavevalue;
			iParametervalue	:=iParametervalue+16#10000;
			istate	:=2;

		(*write Parameter*)
		2:	fbParameterinterface(iParameternumber	:=iParametergroup+16#200,
							iParametervalue		:=iParametervalue,
							stParameterBuffer		:=stParameterBuffer,
							bParametermode		:=TRUE,
							bCycleMode			:=bCycleMode,
							bStart				:=TRUE);
			IF (NOT fbParameterinterface.bBusy) OR bCycleMode THEN
				IF fbParameterinterface.bErr THEN
					bErr			:=TRUE;
					IF fbParameterinterface.iErrornumber =1 THEN
						iErrornumber	:=ERROR_ASI_COMM_ERROR;
					ELSE
						FOR iErrCounter:=2 TO 4 DO
							IF ((SHR(fbParameterinterface.iErrornumber,iErrCounter-2)) AND 16#2000)<>0 THEN
								iErrornumber :=iErrCounter;
							END_IF
						END_FOR
					END_IF
					istate	:=10;
				ELSE
					iParameterReadValue	:=fbParameterinterface.iParameterReadvalue;
					istate	:=3;
				END_IF
			END_IF

		(*read Parametervalue*)
		3:	iReadValue	:=DWORD_TO_WORD(iParameterReadValue);
			IF (NOT bStart) OR (NOT bCycleMode) THEN
				fbParameterinterface(bStart			:=FALSE,
								stParameterBuffer	:=stParameterBuffer);
				IF (NOT fbParameterinterface.bBusy) THEN
					istate	:=10;
				END_IF
			ELSE
				istate	:=1;
			END_IF

			(*Quit*)
		10:	bBusy	:=FALSE;
			IF (NOT bStart) THEN
				istate	:=0;
			END_IF

	ELSE
		;
	END_CASE
END_FUNCTION_BLOCK

(* POU IOF_CAN_Layer2Command, ST *)
FUNCTION_BLOCK IOF_CAN_Layer2Command
VAR_INPUT
	NETID			: T_AmsNetId;
	DEVICEID		: UDINT;
	LEN			: UDINT;
	SRCADDR	: DWORD;
	START			: BOOL;
	TMOUT		: TIME := DEFAULT_ADS_TIMEOUT;
END_VAR
VAR_OUTPUT
	BUSY			: BOOL;
	ERR			: BOOL;
	ERRID			: UDINT;
END_VAR
VAR
	ADSWRITE1	: ADSWRITE;
	RisingEdge	: R_TRIG;
	FallingEdge	: F_TRIG;
END_VAR
RisingEdge(CLK:=START);
IF RisingEdge.Q THEN
	BUSY := TRUE;
	ERR := FALSE;
	ERRID := 0;

	IF ( DEVICEID > 0 ) AND ( MEMSET( SRCADDR, 0, LEN ) > 0 ) THEN
		ADSWRITE1(		NETID:=NETID,
						PORT:= AMSPORT_R0_IO,
						IDXGRP:= 16#00005000 +DEVICEID,
						IDXOFFS:= 16#FFFF0100,
						LEN:= LEN,
						SRCADDR:= SRCADDR,
						WRITE:=TRUE,
						TMOUT:= TMOUT );
	ELSE
		BUSY := FALSE;
		ERR := TRUE;
		ERRID := 1798; (* invalid parameter value *)
		RETURN;
	END_IF
ELSE
	ADSWRITE1( Write:=FALSE);
END_IF


FallingEdge( CLK := ADSWRITE1.BUSY );
IF FallingEdge.Q THEN
	BUSY := FALSE;
	ERR := ADSWRITE1.ERR;
	ERRID := ADSWRITE1.ERRID;
END_IF
END_FUNCTION_BLOCK

(* POU IOF_DeviceReset, ST *)
FUNCTION_BLOCK IOF_DeviceReset
VAR_INPUT
	NETID		: T_AmsNetId;
	DEVICEID	: UDINT;
	RESET		: BOOL;
	TMOUT		: TIME := DEFAULT_ADS_TIMEOUT;
END_VAR
VAR_OUTPUT
	BUSY		: BOOL;
	ERR			: BOOL;
	ERRID		: UDINT;
END_VAR
{library private}
VAR
	ADSWRTCTL1	: ADSWRTCTL := ( PORT := AMSPORT_R0_IO, ADSSTATE := ADSSTATE_RESET, DEVSTATE := 0 );
	RisingEdge	: R_TRIG;
	state		: BYTE;
END_VAR
RisingEdge(CLK:=RESET);
IF RisingEdge.Q THEN
	state := 1;
END_IF
CASE state OF
	0:;(* idle state *)
	1:
		BUSY := TRUE;
		ERR := FALSE;
		ERRID := 0;
		IF ( DeviceId > 0 ) THEN(* if DeviceId=0xAFFE => reset all devices else reset only one device  *)
			ADSWRTCTL1( Write:=FALSE );
			ADSWRTCTL1( NETID := NETID, LEN := SIZEOF( DEVICEID ), SRCADDR := ADR( DEVICEID ), Write := TRUE, TMOUT := TMOUT );
			state := 2;
		ELSE
			ERR := TRUE;
			ERRID := 16#706; (* Parameter value not correct! *)
			state := 100;
		END_IF
	2:
		ADSWRTCTL1( Write:=FALSE, BUSY=>BUSY, ERR=>ERR, ERRID=>ERRID );
		IF NOT BUSY THEN
			state := 0;
		END_IF
	100:(* error state *)
		BUSY := FALSE;
		state := 0;
END_CASE
END_FUNCTION_BLOCK

(* POU IOF_GetBoxAddrByName, ST *)
FUNCTION_BLOCK IOF_GetBoxAddrByName
VAR_INPUT
	NETID		: T_AmsNetId;
	DEVICEID	: UDINT;
	BOXNAME		: T_MaxString;
	START		: BOOL;
	TMOUT		: TIME := DEFAULT_ADS_TIMEOUT;
END_VAR
VAR_OUTPUT
	BUSY		: BOOL;
	ERR			: BOOL;
	ERRID		: UDINT;
	BOXADDR		: UINT;
END_VAR
{library private}
VAR
	ADSRDWRTEX1	: ADSRDWRTEX := ( PORT:= AMSPORT_R0_IO, IDXOFFS:= 16#00000004 );
	RisingEdge	: R_TRIG;
	state		: BYTE;
END_VAR
RisingEdge(CLK:=START);
IF RisingEdge.Q THEN
	state := 1;
END_IF
CASE state OF
	0:;(* idle state *)
	1:
		BUSY := TRUE;
		ERR:= FALSE;
		ERRID := 0;
		BOXADDR:=0;
		IF ( DEVICEID > 0 ) AND ( BOXNAME <> '' ) THEN
			ADSRDWRTEX1( WRTRD:=FALSE );
			ADSRDWRTEX1(	NETID:=NETID, IDXGRP:= 16#00005000 + DEVICEID,
							WRITELEN:=LEN( BOXNAME )+1, READLEN:=SIZEOF( BOXADDR ),
							SRCADDR:=ADR( BOXNAME ), DESTADDR:= ADR( BOXADDR ),
							WRTRD:=TRUE, TMOUT:= TMOUT );
			state := 2;
		ELSE
			ERR := TRUE;
			ERRID := 16#706; (* Parameter value not correct! *)
			state := 100;
		END_IF
	2:
		ADSRDWRTEX1( WRTRD:=FALSE, BUSY=>BUSY, ERR=>ERR, ERRID=>ERRID );
		IF NOT BUSY THEN
			IF NOT ERR THEN
				IF ( ADSRDWRTEX1.COUNT_R = SIZEOF( BOXADDR ) ) THEN (* check the read data length *)
					;(* OK *)
				ELSE
					ERR := TRUE;
					ERRID := 16#70B; (* 1803 invalid parameter value(s) *)
				END_IF
			END_IF
			state := 0;
		END_IF
	100:(* error state *)
		BUSY := FALSE;
		state := 0;
END_CASE
END_FUNCTION_BLOCK

(* POU IOF_GetBoxAddrByNameEx, ST *)
FUNCTION_BLOCK IOF_GetBoxAddrByNameEx
VAR_INPUT
	NETID		: T_AmsNetId;
	DEVICENAME	: T_MaxString;
	BOXNAME		: T_MaxString;
	START		: BOOL;
	TMOUT		: TIME := DEFAULT_ADS_TIMEOUT;
END_VAR
VAR_OUTPUT
	BUSY		: BOOL;
	ERR			: BOOL;
	ERRID		: UDINT;
	BOXADDR		: UINT;
END_VAR
{library private}
VAR
	ADSRDWRTEX1	: ADSRDWRTEX := ( PORT:= AMSPORT_R0_IO, IDXOFFS:= 16#00000004 );
	RisingEdge	: R_TRIG;
	state		: BYTE;
	StrBuff		: STRING(512);
END_VAR
RisingEdge(CLK:=START);
IF RisingEdge.Q THEN
	state := 1;
END_IF
CASE state OF
	0:;(* idle state *)
	1:
		BUSY:= TRUE;
		ERR := FALSE;
		ERRID := 0;
		BOXADDR:=0;
		IF ( DeviceName <> '' ) AND ( BoxName <> '' ) THEN
			StrBuff:=CONCAT( DeviceName, '.' );
			StrBuff:=CONCAT( StrBuff, BoxName );
			ADSRDWRTEX1( WRTRD:=FALSE );
			ADSRDWRTEX1( NETID:=NETID, IDXGRP:= 16#00005000,
						WRITELEN:= LEN( StrBuff )+1, READLEN:=SIZEOF( BOXADDR ),
						SRCADDR:=ADR( StrBuff ), DESTADDR:= ADR( BOXADDR ),
						WRTRD:=TRUE, TMOUT:= TMOUT );
			state := 2;
		ELSE
			ERR := TRUE;
			ERRID := 16#706; (* Parameter value not correct! *)
			state := 100;
		END_IF
	2:
		ADSRDWRTEX1( WRTRD:=FALSE, BUSY=>BUSY, ERR=>ERR, ERRID=>ERRID );
		IF NOT BUSY THEN
			IF NOT ERR THEN
				IF ( ADSRDWRTEX1.COUNT_R = SIZEOF( BOXADDR ) ) THEN (* check the read data length *)
					;(* OK*)
				ELSE
					ERR := TRUE;
					ERRID := 16#70B; (* 1803 invalid parameter value(s) *)
				END_IF
			END_IF
			state := 0;
		END_IF
	100:(* error state *)
		BUSY := FALSE;
		state := 0;
END_CASE
END_FUNCTION_BLOCK

(* POU IOF_GetBoxCount, ST *)
FUNCTION_BLOCK IOF_GetBoxCount
VAR_INPUT
	NETID		: T_AmsNetId;
	DEVICEID	: UDINT;
	START		: BOOL;
	TMOUT		: TIME := DEFAULT_ADS_TIMEOUT;
END_VAR
VAR_OUTPUT
	BUSY		: BOOL;
	ERR			: BOOL;
	ERRID		: UDINT;
	BOXCOUNT	: UDINT;
END_VAR
{library private}
VAR
	ADSREADEX1	: ADSREADEX := ( PORT:= AMSPORT_R0_IO, IDXOFFS:= 16#00000002 );
	RisingEdge	: R_TRIG;
	state		: BYTE;
END_VAR
RisingEdge(CLK:=START);
IF RisingEdge.Q THEN
	state := 1;
END_IF
CASE state OF
	0:;(* idle state *)
	1:
		BUSY := TRUE;
		ERR:= FALSE;
		ERRID := 0;
		BOXCOUNT:=0;
		IF DEVICEID > 0 THEN
			ADSREADEX1( READ:=FALSE );
			ADSREADEX1( NETID:=NETID, IDXGRP:= 16#00005000 +DEVICEID,
						LEN:= SIZEOF( BOXCOUNT ), DESTADDR:= ADR( BOXCOUNT ),
						READ:=TRUE, TMOUT:= TMOUT );
			state := 2;
		ELSE
			ERR := TRUE;
			ERRID :=16#706;(* Parameter value not correct! *)
			state := 100;
		END_IF
	2:
		ADSREADEX1( READ:=FALSE, BUSY=>BUSY, ERR=>ERR, ERRID=>ERRID );
		IF NOT BUSY THEN
			IF NOT ERR THEN
				IF ( ADSREADEX1.COUNT_R <= SIZEOF( BOXCOUNT ) ) THEN
					;(*OK=> ChristophC: 13.08.2010-> Some 15xx builds and all TwinCAT 20xx and higher are returning only 2 bytes. Workaround: Allow 2 bytes as return length too. *)
				ELSE
					ERR := TRUE;
					ERRID := 16#70B; (* 1803 invalid parameter value(s) *)
				END_IF
			END_IF
			state := 0;
		END_IF
	100:(* error state *)
		BUSY := FALSE;
		state := 0;
END_CASE
END_FUNCTION_BLOCK

(* POU IOF_GetBoxNameByAddr, ST *)
FUNCTION_BLOCK IOF_GetBoxNameByAddr
VAR_INPUT
	NETID		: T_AmsNetId;
	DEVICEID	: UDINT;
	BOXADDR		: UINT;
	START		: BOOL;
	TMOUT		: TIME := DEFAULT_ADS_TIMEOUT;
END_VAR
VAR_OUTPUT
	BUSY		: BOOL;
	ERR			: BOOL;
	ERRID		: UDINT;
	BOXNAME		: T_MaxString;
END_VAR
{library private}
VAR
	ADSRDWRTEX1	: ADSRDWRTEX := ( PORT:= AMSPORT_R0_IO, IDXOFFS:= 16#00000003 );
	RisingEdge	: R_TRIG;
	state		: BYTE;
END_VAR
RisingEdge(CLK:=START);
IF RisingEdge.Q THEN
	state := 1;
END_IF
CASE state OF
	0:;(* idle state *)
	1:
		BUSY:=TRUE;
		ERR:=FALSE;
		ERRID := 0;
		MEMSET( ADR( BOXNAME ), 0, SIZEOF( BOXNAME ) );
		IF ( DEVICEID > 0 ) AND ( BOXADDR > 0 ) THEN
			ADSRDWRTEX1( WRTRD:=FALSE );
			ADSRDWRTEX1(NETID:=NETID, IDXGRP:= 16#00005000 + DEVICEID,
						WRITELEN:= SIZEOF( BOXADDR ), READLEN:=SIZEOF( BOXNAME ) - 1, (* saves termination byte *)
						SRCADDR:=ADR( BOXADDR ), DESTADDR:= ADR( BOXNAME ),
						WRTRD:=TRUE, TMOUT:= TMOUT );
			state := 2;
		ELSE
			ERR := TRUE;
			ERRID := 16#706;(* Parameter value not correct! *)
			state := 100;
		END_IF
	2:
		ADSRDWRTEX1( WRTRD:=FALSE, BUSY=>BUSY, ERR=>ERR, ERRID=>ERRID );
		IF NOT BUSY THEN
			state := 0;
		END_IF
	100:(* error state *)
		BUSY := FALSE;
		state := 0;
END_CASE
END_FUNCTION_BLOCK

(* POU IOF_GetBoxNetId, ST *)
FUNCTION_BLOCK IOF_GetBoxNetId
VAR_INPUT
	NETID		: T_AmsNetId;
	DEVICEID	: UDINT;
	BOXADDR		: WORD;
	START		: BOOL;
	TMOUT		: TIME := DEFAULT_ADS_TIMEOUT;
END_VAR
VAR_OUTPUT
	BUSY		: BOOL;
	ERR			: BOOL;
	ERRID		: UDINT;
	BoxNetId	: T_AmsNetId;
END_VAR
{library private}
VAR
	ADSRDWRTEX1	: ADSRDWRTEX := ( PORT:= AMSPORT_R0_IO, IDXOFFS:= 16#00000006 );
	RisingEdge	: R_TRIG;
	state		: BYTE;
	tmpNetId	: ARRAY[0..5] OF BYTE;
END_VAR
RisingEdge( CLK:=START );
IF RisingEdge.Q THEN
	state := 1;
END_IF
CASE state OF
	0:;(* idle state *)
	1:
		BUSY := TRUE;
		ERR := FALSE;
		ERRID := 0;
		BoxNetId := '';
		MEMSET( ADR( tmpNetId ), 0, SIZEOF( tmpNetId ) );
		IF ( DEVICEID > 0 ) AND ( BOXADDR > 0 ) THEN
			ADSRDWRTEX1( WRTRD:= FALSE );
			ADSRDWRTEX1( NETID:=NETID, IDXGRP:= 16#00005000 + DEVICEID,
						WRITELEN:= SIZEOF( BOXADDR ), READLEN:= SIZEOF( tmpNetId ),
						SRCADDR:= ADR( BOXADDR ), DESTADDR:= ADR( tmpNetId ),
						WRTRD:= TRUE, TMOUT:= TMOUT );
			state := 2;
		ELSE
			ERR := TRUE;
			ERRID :=16#706;	(* Parameter value not correct! *)
			state := 100;
		END_IF
	2:
		ADSRDWRTEX1( WRTRD:= FALSE, BUSY=>BUSY, ERR=>ERR, ERRID=>ERRID );
		IF NOT BUSY THEN
			IF NOT ERR THEN
				IF ( ADSRDWRTEX1.COUNT_R = SIZEOF( tmpNetId ) ) THEN (* check the read data length *)
					BoxNetId := F_CreateAmsNetId( tmpNetId );(* OK *)
				ELSE
					ERR := TRUE;
					ERRID := 16#70B; (* 1803 invalid parameter value(s) *)
				END_IF
			END_IF
			state := 0;
		END_IF
	100:(* error state *)
		BUSY:= FALSE;
		state := 0;
END_CASE
END_FUNCTION_BLOCK

(* POU IOF_GetDeviceCount, ST *)
FUNCTION_BLOCK IOF_GetDeviceCount
VAR_INPUT
	NETID		: T_AmsNetId;
	START		: BOOL;
	TMOUT		: TIME := DEFAULT_ADS_TIMEOUT;
END_VAR
VAR_OUTPUT
	BUSY		: BOOL;
	ERR			: BOOL;
	ERRID		: UDINT;
	DEVICECOUNT	: UDINT;
END_VAR
{library private}
VAR
	ADSREADEX1	: ADSREADEX := ( PORT:= AMSPORT_R0_IO, IDXGRP:= 16#00005000, IDXOFFS:= 16#00000002 );
	RisingEdge	: R_TRIG;
	state 		: BYTE;
END_VAR
RisingEdge(CLK:=START);
IF RisingEdge.Q THEN
	state := 1;
END_IF
CASE state OF
	0:;(* idle state *)
	1:
		BUSY := TRUE;
		ERR := FALSE;
		ERRID := 0;
		DEVICECOUNT := 0;
		ADSREADEX1( READ:=FALSE );
		ADSREADEX1( NETID:=NETID, LEN:= SIZEOF( DEVICECOUNT ), DESTADDR:= ADR( DEVICECOUNT ), READ:=TRUE, TMOUT:= TMOUT );
		state := 2;
	2:
		ADSREADEX1( READ:=FALSE, BUSY=>BUSY, ERR=>ERR, ERRID=>ERRID );
		IF NOT BUSY THEN
			IF NOT ERR THEN
				IF ( ADSREADEX1.COUNT_R = SIZEOF( DEVICECOUNT ) ) THEN (* check the read data length *)
					;(* OK *)
				ELSE
					ERR := TRUE;
					ERRID := 16#70B; (* 1803 invalid parameter value(s) *)
				END_IF
			END_IF
			state := 0;
		END_IF
END_CASE
END_FUNCTION_BLOCK

(* POU IOF_GetDeviceIDByName, ST *)
FUNCTION_BLOCK IOF_GetDeviceIDByName
VAR_INPUT
	NETID		: T_AmsNetId;
	DEVICENAME	: T_MaxString;
	START		: BOOL;
	TMOUT		: TIME := DEFAULT_ADS_TIMEOUT;
END_VAR
VAR_OUTPUT
	BUSY		: BOOL;
	ERR			: BOOL;
	ERRID		: UDINT;
	DEVICEID	: UDINT;
END_VAR
{library private}
VAR
	ADSRDWRTEX1	: ADSRDWRTEX := ( PORT:= AMSPORT_R0_IO, IDXGRP:= 16#00005000, IDXOFFS:= 16#00000003 );
	RisingEdge	: R_TRIG;
	state		: BYTE;
END_VAR
RisingEdge(CLK:=START);
IF RisingEdge.Q THEN
	state := 1;
END_IF
CASE state OF
	0:;(* state idle *)
	1:
		BUSY := TRUE;
		ERR := FALSE;
		ERRID := 0;
		DEVICEID:=0;
		IF ( DeviceName <> '' ) THEN
			ADSRDWRTEX1( WRTRD:=FALSE );
			ADSRDWRTEX1(	NETID:=NETID, WRITELEN:= LEN( DEVICENAME )+1, READLEN:=SIZEOF( DEVICEID ),
							SRCADDR:=ADR( DEVICENAME ), DESTADDR:= ADR( DEVICEID ),
							WRTRD:=TRUE, TMOUT:= TMOUT );
			state := 2;
		ELSE
			ERR := TRUE;
			ERRID :=16#706;	(* Parameter value not correct! *)
			state := 100;
		END_IF
	2:
		ADSRDWRTEX1( WRTRD:=FALSE, BUSY=>BUSY, ERR=>ERR, ERRID=>ERRID );
		IF NOT BUSY THEN
			IF NOT ERR THEN
				IF ( ADSRDWRTEX1.COUNT_R =  SIZEOF( DEVICEID ) ) THEN (* check the read data length *)
					;(* OK *)
				ELSE
					ERR := TRUE;
					ERRID := 16#70B; (* 1803 invalid parameter value(s) *)
				END_IF
			END_IF
			state := 0;
		END_IF
	100:(* error state *)
		BUSY:= FALSE;
		state := 0;
END_CASE
END_FUNCTION_BLOCK

(* POU IOF_GetDeviceIDs, ST *)
FUNCTION_BLOCK IOF_GetDeviceIDs
VAR_INPUT
	NETID		: T_AmsNetId;
	LEN			: UDINT;
	DESTADDR	: DWORD;
	START		: BOOL;
	TMOUT		: TIME := DEFAULT_ADS_TIMEOUT;
END_VAR
VAR_OUTPUT
	BUSY		: BOOL;
	ERR			: BOOL;
	ERRID		: UDINT;
END_VAR
{library private}
VAR
	ADSREADEX1	: ADSREADEX := ( PORT:= AMSPORT_R0_IO, IDXGRP:= 16#00005000, IDXOFFS:= 16#00000001 );
	RisingEdge	: R_TRIG;
	state 		: BYTE;
END_VAR
RisingEdge(CLK:=START);
IF RisingEdge.Q THEN
	state := 1;
END_IF
CASE state OF
	0:;(* idle state *)
	1:
		BUSY := TRUE;
		ERR := FALSE;
		ERRID := 0;
		IF ( MEMSET( DESTADDR, 0, LEN ) > 0 ) THEN
			ADSREADEX1( READ:=FALSE);
			ADSREADEX1( NETID:=NETID, LEN:= LEN, DESTADDR:= DESTADDR, READ:=TRUE, TMOUT:= TMOUT );
			state := 2;
		ELSE
			ERR := TRUE;
			ERRID := 16#706;	(* Parameter value not correct! *)
			state := 100;
		END_IF
	2:
		ADSREADEX1( READ:=FALSE, BUSY=>BUSY, ERR=>ERR, ERRID=>ERRID );
		IF NOT BUSY THEN
			state := 0;
		END_IF
	100:(* error state *)
		BUSY := FALSE;
		state := 0;
END_CASE
END_FUNCTION_BLOCK

(* POU IOF_GetDeviceInfoByName, ST *)
FUNCTION_BLOCK IOF_GetDeviceInfoByName
VAR_INPUT
	NETID			: T_AmsNetId;
	DEVICENAME		: T_MaxString;
	START			: BOOL;
	TMOUT			: TIME := DEFAULT_ADS_TIMEOUT;
END_VAR
VAR_OUTPUT
	BUSY			: BOOL;
	ERR				: BOOL;
	ERRID			: UDINT;
	DEVICEID		: UDINT;
	DEVICENETID		: T_AmsNetId;
END_VAR
{library private}
VAR
	ADSRDWRTEX1		: ADSRDWRTEX := ( PORT:= AMSPORT_R0_IO, IDXGRP:= 16#00005000, IDXOFFS:= 16#00000003 );
	ADSREADEX1		: ADSREADEX := ( PORT:= AMSPORT_R0_IO, IDXOFFS:= 16#00000005 );
	tmpNetId		: ARRAY[0..5] OF BYTE;
	state			: BYTE;
	RisingEdge		: R_TRIG;
END_VAR
RisingEdge(CLK:=START);
IF RisingEdge.Q THEN
	state 	:= 1;
END_IF

CASE state OF
	0:; (*do nothing*)
	1:
		BUSY := TRUE;
		ERR := FALSE;
		ERRID := 0;
		DEVICEID:=0;
		DEVICENETID := '';
		IF ( DeviceName <> '' ) THEN
			ADSRDWRTEX1( WRTRD:=FALSE); (*fb reset*)
			ADSRDWRTEX1(NETID:=NETID, WRITELEN:= LEN(DEVICENAME)+1, READLEN:=SIZEOF(DEVICEID),
						SRCADDR:=ADR(DEVICENAME), DESTADDR:= ADR(DEVICEID), WRTRD:=TRUE, TMOUT:= TMOUT);
			state := state + 1;

		ELSE
			ERR := TRUE;
			ERRID :=16#706;	(* Parameter value not correct! *)
			state := 100;
		END_IF

	2:
		ADSRDWRTEX1( WRTRD:=FALSE);
		IF NOT ADSRDWRTEX1.BUSY THEN
			IF NOT ADSRDWRTEX1.ERR  THEN
				IF ( DEVICEID <> 0 ) AND  ( ADSRDWRTEX1.COUNT_R = ADSRDWRTEX1.READLEN ) THEN
					ADSREADEX1( READ:=FALSE);
					ADSREADEX1( NETID:=NETID, IDXGRP:= 16#00005000 + DEVICEID,
								LEN:= SIZEOF(tmpNetId), DESTADDR:= ADR(tmpNetId),
								READ:=TRUE, TMOUT:= TMOUT );
					state := state + 1;
				ELSE
					BUSY:= FALSE;
					ERR := TRUE;
					ERRID := 16#70B; (* 1803 invalid parameter value(s) *)
					state := 0;
				END_IF
			ELSE
				BUSY:= FALSE;
				ERR := TRUE;
				ERRID := ADSRDWRTEX1.ERRID;
				state := 0;
			END_IF
		END_IF
	3:
		ADSREADEX1( READ:=FALSE);
		IF NOT ADSREADEX1.BUSY THEN
			state := 0;
			BUSY:= FALSE;
			ERR := ADSREADEX1.ERR;
			ERRID := ADSREADEX1.ERRID;

			IF ( ( NOT ERR ) AND ( ADSREADEX1.COUNT_R <> ADSREADEX1.LEN ) ) THEN (* check the read data length *)
				ERR := TRUE;
				ERRID := 16#70B; (* 1803 invalid parameter value(s) *)
			ELSE
				DeviceNetId := F_CreateAmsNetId( tmpNetid );
			END_IF
		END_IF

100:(* error step *)
	BUSY := FALSE;
	state := 0;

END_CASE
END_FUNCTION_BLOCK

(* POU IOF_GetDeviceName, ST *)
FUNCTION_BLOCK IOF_GetDeviceName
VAR_INPUT
	NETID		: T_AmsNetId;
	DEVICEID	: UDINT;
	START		: BOOL;
	TMOUT		: TIME := DEFAULT_ADS_TIMEOUT;
END_VAR
VAR_OUTPUT
	BUSY		: BOOL;
	ERR			: BOOL;
	ERRID		: UDINT;
	DEVICENAME	: T_MaxString;
END_VAR
{library private}
VAR
	ADSREADEX1	: ADSREADEX := ( PORT:= AMSPORT_R0_IO, IDXOFFS:= 16#00000001 );
	RisingEdge	: R_TRIG;
	state		: BYTE;
END_VAR
RisingEdge(CLK:=START);
IF RisingEdge.Q THEN
	state := 1;
END_IF
CASE state OF
	0:;(* idle state *)
	1:
		BUSY := TRUE;
		ERR := FALSE;
		ERRID := 0;
		MEMSET( ADR( DEVICENAME ), 0, SIZEOF( DEVICENAME ) );
		IF ( DEVICEID > 0 ) THEN
			ADSREADEX1( READ:=FALSE );
			ADSREADEX1( NETID:=NETID, IDXGRP:= 16#00005000 + DEVICEID,
						LEN:= SIZEOF( DEVICENAME ) - 1, (* save string termination *)
						DESTADDR:= ADR( DEVICENAME ), READ:=TRUE, TMOUT:= TMOUT );
			state := 2;
		ELSE
			ERR:=TRUE;
			ERRID :=16#706;	(*	Parameter value not correct!	*)
			state := 100;
		END_IF
	2:
		ADSREADEX1( READ:=FALSE, BUSY=>BUSY, ERR=>ERR, ERRID=>ERRID );
		IF NOT BUSY THEN
			state := 0;
		END_IF
	100:(* error state *)
		BUSY:=FALSE;
		state := 0;
END_CASE
END_FUNCTION_BLOCK

(* POU IOF_GetDeviceType, ST *)
FUNCTION_BLOCK IOF_GetDeviceType
VAR_INPUT
	NETID			: T_AmsNetId;
	DEVICEID		: UDINT;
	START			: BOOL;
	TMOUT			: TIME := DEFAULT_ADS_TIMEOUT;
END_VAR
VAR_OUTPUT
	BUSY			: BOOL;
	ERR				: BOOL;
	ERRID			: UDINT;
	IODeviceType	: IODEVICETYPES;
END_VAR
{library private}
VAR
	ADSREADEX1		: ADSREADEX := ( PORT:= AMSPORT_R0_IO, IDXOFFS:= 16#00000007 );
	RisingEdge		: R_TRIG;
	state			: BYTE;
	tmpDeviceType	: WORD:=0;
END_VAR
RisingEdge( CLK:=START );
IF RisingEdge.Q THEN
	state := 1;
END_IF
CASE state OF
	0:;(* idle state *)
	1:
		BUSY := TRUE;
		ERR:= FALSE;
		ERRID := 0;
		IODeviceType := IODEVICETYPE_UNKNOWN;
		tmpDeviceType := 0;
		IF ( DEVICEID > 0 ) THEN
			ADSREADEX1( READ:=FALSE );
			ADSREADEX1( NETID:=NETID, IDXGRP:= 16#00005000 + DEVICEID,
						LEN:= SIZEOF( tmpDeviceType ), DESTADDR:= ADR( tmpDeviceType ),
						READ:=TRUE, TMOUT:= TMOUT );
			state := 2;
		ELSE
			ERR := TRUE;
			ERRID := 16#706;	(* Parameter value not correct! *)
			state := 100;
		END_IF
	2:
		ADSREADEX1( READ:=FALSE, BUSY=>BUSY, ERR=>ERR, ERRID=>ERRID );
		IF NOT BUSY THEN
			IF NOT ERR THEN
				IF ( ADSREADEX1.COUNT_R = SIZEOF( tmpDeviceType ) ) THEN
					IODeviceType := tmpDeviceType;(* OK *)
				ELSE
					;(* error? *)
				END_IF
			END_IF
			state := 0;
		END_IF
	100:(* error state *)
		BUSY := FALSE;
		state := 0;
END_CASE
END_FUNCTION_BLOCK

(* POU IOF_LB_BreakLocationTest, ST *)
FUNCTION_BLOCK IOF_LB_BreakLocationTest
VAR_INPUT
	NETID			: T_AmsNetId;
	DEVICEID		: UDINT;
	START			: BOOL;
	TMOUT		: TIME := DEFAULT_ADS_TIMEOUT;
END_VAR
VAR_OUTPUT
	BUSY			: BOOL;
	ERR			: BOOL;
	ERRID			: UDINT;
	BREAK		: BOOL;
	BOXNO		: WORD;
END_VAR
VAR
	ADSREADEX1	: ADSREADEX;
	RisingEdge	: R_TRIG;
	FallingEdge	: F_TRIG;
	TestData		: ARRAY[0..3] OF BYTE;
END_VAR
RisingEdge(CLK:=START);
IF RisingEdge.Q THEN
	BUSY := TRUE;
	ERR := FALSE;
	ERRID := 0;
	BREAK:=FALSE;
	BOXNO:=0;
	MEMSET( ADR( TestData ), 0 , SIZEOF( TestData ) );

	ADSREADEX1(		NETID:=NETID,
					PORT:= AMSPORT_R0_IO,
					IDXGRP:= 16#00005000 +DEVICEID,
					IDXOFFS:= 16#FFFF0100,
					LEN:= SIZEOF(TestData),(*4 Byte*)
					DESTADDR:= ADR(TestData),
					READ:=TRUE,
					TMOUT:= TMOUT);
ELSE
	ADSREADEX1( READ:=FALSE);
END_IF


FallingEdge( CLK := ADSREADEX1.BUSY );
IF FallingEdge.Q THEN
	BUSY := FALSE;

	ERR := ADSREADEX1.ERR;
	ERRID := ADSREADEX1.ERRID;

	IF TestData[1]=0 THEN(*no break*)
		BOXNO:=TestData[0];(*break location ->Box*)
		BREAK:=FALSE;
	ELSIF TestData[0]=1 AND TestData[1]=16#FF THEN(*not be localize*)
		BOXNO:=0;
		BREAK:=TRUE;
	ELSIF TestData[1]=16#FF THEN(*can localize*)
		BOXNO:=-TestData[0];
		BREAK:=TRUE;
	END_IF

	IF ( ( NOT ERR ) AND ( ADSREADEX1.COUNT_R <> ADSREADEX1.LEN ) ) THEN
		ERR := TRUE;
		ERRID := 16#70B; (* 1803 invalid parameter value(s) *)
	END_IF

END_IF
END_FUNCTION_BLOCK

(* POU IOF_LB_ParityCheck, ST *)
FUNCTION_BLOCK IOF_LB_ParityCheck
VAR_INPUT
	NETID			: T_AmsNetId;
	DEVICEID		: UDINT;
	LEN			: UDINT;
	DESTADDR	: DWORD;
	START			: BOOL;
	TMOUT		: TIME := DEFAULT_ADS_TIMEOUT;
END_VAR
VAR_OUTPUT
	BUSY			: BOOL;
	ERR			: BOOL;
	ERRID			: UDINT;
END_VAR
VAR
	ADSREADEX1	: ADSREADEX;
	RisingEdge	: R_TRIG;
	FallingEdge	: F_TRIG;
END_VAR
RisingEdge(CLK:=START);
IF RisingEdge.Q THEN
	BUSY := TRUE;
	ERR:= FALSE;
	ERRID := 0;

	IF ( DEVICEID > 0 ) AND ( MEMSET( DESTADDR, 0, LEN ) > 0 ) THEN
		ADSREADEX1(		NETID:=NETID,
						PORT:= AMSPORT_R0_IO,
						IDXGRP:= 16#00005000 + DEVICEID,
						IDXOFFS:= 16#FFFF0200,
						LEN:= LEN,
						DESTADDR:=DESTADDR,
						READ:=TRUE,
						TMOUT:= TMOUT);
	ELSE
		BUSY := FALSE;
		ERR:=TRUE;
		ERRID :=16#706;(* Parameter value not correct! *)
		RETURN;
	END_IF
ELSE
	ADSREADEX1( READ:=FALSE);
END_IF


FallingEdge( CLK := ADSREADEX1.BUSY );
IF FallingEdge.Q THEN
	BUSY := FALSE;
	ERR := ADSREADEX1.ERR;
	ERRID := ADSREADEX1.ERRID;
END_IF
END_FUNCTION_BLOCK

(* POU IOF_LB_ParityCheckWithReset, ST *)
FUNCTION_BLOCK IOF_LB_ParityCheckWithReset
VAR_INPUT
	NETID			: T_AmsNetId;
	DEVICEID		: UDINT;
	LEN			: UDINT;
	DESTADDR	: DWORD;
	START			: BOOL;
	TMOUT		: TIME := DEFAULT_ADS_TIMEOUT;
END_VAR
VAR_OUTPUT
	BUSY			: BOOL;
	ERR			: BOOL;
	ERRID			: UDINT;
END_VAR
VAR
	ADSREADEX1	: ADSREADEX;
	RisingEdge	: R_TRIG;
	FallingEdge	: F_TRIG;
END_VAR
RisingEdge(CLK:=START);
IF RisingEdge.Q THEN
	BUSY := TRUE;
	ERR := FALSE;
	ERRID := 0;

	IF ( DEVICEID > 0 ) AND ( MEMSET( DESTADDR, 0, LEN ) > 0 ) THEN
		ADSREADEX1(		NETID:=NETID,
						PORT:= AMSPORT_R0_IO,
						IDXGRP:= 16#00005000 +DEVICEID,
						IDXOFFS:= 16#FFFF0300,
						LEN:= LEN,
						DESTADDR:= DESTADDR,
						READ:=TRUE,
						TMOUT:= TMOUT );
	ELSE
		BUSY := FALSE;
		ERR:=TRUE;
		ERRID :=16#706;(* Parameter value not correct! *)
		RETURN;
	END_IF
ELSE
	ADSREADEX1( READ:=FALSE);
END_IF

FallingEdge( CLK := ADSREADEX1.BUSY );
IF FallingEdge.Q THEN
	BUSY := FALSE;
	ERR := ADSREADEX1.ERR;
	ERRID := ADSREADEX1.ERRID;
END_IF
END_FUNCTION_BLOCK

(* POU IOF_SER_DRIVE_Backup, ST *)
FUNCTION_BLOCK IOF_SER_DRIVE_Backup
VAR_INPUT
	bCheck				: BOOL;
	bBackup				: BOOL;
	bRestore				: BOOL;
	bCRCEnable			: BOOL			:= TRUE;
	bStdBackupList		: BOOL 			:= TRUE;
	sNetId 					: T_AmsNetId;
	nPort					: UINT;
	sComment			: T_MaxString;
	ePath					: E_OpenPath 	:= PATH_BOOTPATH;
	sPathName			: T_MaxString 	:= 'DRIVEPAR.BIN';
	tTimeout				: TIME := DEFAULT_ADS_TIMEOUT;
END_VAR
VAR_OUTPUT
	bBusy					: BOOL;
	bError					: BOOL;
	nErrId					: UDINT;
	bCheckOK				: BOOL;
(*	Function block specific error codes:
	16#1005 = false backup parameter type 
	16#1006 = backup list was not IDN 192

*)
END_VAR
VAR CONSTANT
	iVALUE					: DINT := 0;
END_VAR
VAR
	ReadSercosParam			: IOF_SER_IDN_Read;
	WriteSercosParam		: IOF_SER_IDN_Write;

	OpenBackupFile			: FB_FileOpen;
	CloseBackupFile			: FB_FileClose;
	ReadBackupFile			: FB_FileRead;
	WriteBackupFile			: FB_FileWrite;

	eState					: E_SercosBackupState;

	sCheckData				: ST_SercosString;
	wCRC16_CCITT			: WORD;
	wCheckSum				: WORD;

	bCheck_I				: BOOL;
	bBackup_I				: BOOL;
	bRestore_I				: BOOL;
	bCheck_L				: BOOL;
	bBackup_L				: BOOL;
	bRestore_L				: BOOL;
	bUpdateCRC				: BOOL;

	bBackupDone				: BOOL;
	bRestoreDone			: BOOL;

	arrList					: ARRAY [0..65535] OF BYTE;
	nListArrIdx				: UINT;
	sListAttrib				: ST_SercosParamAttrib;

	cbLen					: UDINT;
	arrData					: ARRAY [0..65535] OF BYTE;

	nIDN					: UINT;
	nCRCIDN					: UINT := 142;
	bCRCIDNExist			: BOOL;
	bCRCIDNTest				: BOOL := TRUE;
	iIdx					: UINT;

	sParamHeader			: ST_SercosParamHeader;
	cbSize					: UDINT;
	sFileHeader				: ST_SercosFileHeader;
	sParamData				: ST_SercosParamData;

	iActListItem			: UINT;
	iLastListItem			: UINT;
	bEndOfList				: BOOL;

	bFileOpen				: BOOL;
	hFile					: UINT;
	nVersion				: UDINT := 1;
	nRetVal					: UDINT;

	bWrongListType			: BOOL;
	bFileError				: BOOL;
	nFileErrId				: UDINT;
	bIdnError				: BOOL;
	nIdnErrId				: UDINT;
	nIdnAccessId			: UINT;
END_VAR
VAR PERSISTENT
	wSavedCRC16_CCITT		: WORD;
	wSavedCheckSum			: WORD;
	sSavedCheckData			: ST_SercosString;
END_VAR
(* state machine *)
CASE eState OF
	eBkup_IDLE:
		bBusy 		 		:= FALSE;

		(* wait for command *)
		IF bCheck AND bCRCIDNTest AND bCRCEnable THEN
			bError			:= FALSE;
			nErrId			:= 0;
			bFileOpen		:= FALSE;
			bFileError		:= FALSE;
			nFileErrId		:= 0;
			bWrongListType	:= FALSE;
			bIdnError		:= FALSE;
			nIdnErrId		:= 0;
			nIdnAccessId	:= 0;
			bEndOfList		:= FALSE;
			eState 			:= eBkup_READ_IDNLIST_INI;
			bBusy			:= TRUE;
			bCheckOK 		:= FALSE;

		ELSIF (bCheck AND NOT(bCheck_I)) AND bCRCEnable AND bCRCIDNExist THEN
			bError			:= FALSE;
			nErrId			:= 0;
			bFileOpen		:= FALSE;
			bFileError		:= FALSE;
			nFileErrId		:= 0;
			bWrongListType	:= FALSE;
			bIdnError		:= FALSE;
			nIdnErrId		:= 0;
			nIdnAccessId	:= 0;
			bEndOfList		:= FALSE;
			eState 			:= eBkup_CHECK_CRC_ACT;
			bBusy			:= TRUE;
			bCheckOK 		:= FALSE;
			bCheck_I 		:= TRUE;

			ReadSercosParam(bExecute := FALSE);
			ReadSercosParam(
				sNetId 		:= sNetId,
				nIDN		:= nCRCIDN,
				bExecute	:= TRUE,
				nMode		:= iVALUE,
				nPort		:= nPort,
				nAttrib		:= 0,
				cbLen		:= SIZEOF(sCheckData),
				dwDestAddr 	:= ADR(sCheckData),
				tTimeout	:= tTimeout
			);
		ELSE
			IF (bBackup AND NOT(bBackup_I)) OR (bRestore AND NOT(bRestore_I)) THEN
				bBackup_L		:= FALSE;
				bRestore_L		:= FALSE;
				bBusy			:= FALSE;
				bError			:= FALSE;
				nErrId			:= 0;
				bFileOpen		:= FALSE;
				bFileError		:= FALSE;
				nFileErrId		:= 0;
				bWrongListType	:= FALSE;
				bIdnError		:= FALSE;
				nIdnErrId		:= 0;
				nIdnAccessId	:= 0;
				bEndOfList		:= FALSE;
				eState 			:= eBkup_READ_IDNLIST_INI;
				bBusy			:= TRUE;
				bUpdateCRC		:= TRUE;
				bCheckOK 		:= FALSE;

				(* initialize CRC16-CCITT and CheckSum *)
				wSavedCRC16_CCITT 			:= 16#FFFF;
				wSavedCheckSum	  			:= 16#0000;
				sSavedCheckData.iActSize	:= 0;
				sSavedCheckData.sString		:= '';

				IF bBackup AND NOT(bBackup_I) THEN
					(* latch backup request *)
					bBackup_L	:= TRUE;
					bRestore_L	:= FALSE;
					bBackup_I 	:= TRUE;

				ELSIF bRestore AND NOT(bRestore_I) THEN
					(* latch restore request *)
					bBackup_L	:= FALSE;
					bRestore_L	:= TRUE;
					bRestore_I	:= TRUE;
				END_IF
			END_IF
		END_IF

		wCRC16_CCITT 		:= wSavedCRC16_CCITT;
		wCheckSum	 		:= wSavedCheckSum;


	(*** check CRC and CheckSum ***)
	eBkup_CHECK_CRC_ACT:
		ReadSercosParam(bExecute := FALSE);

		IF NOT(ReadSercosParam.bBusy) THEN
			(* not busy anymore *)
			bError	:= ReadSercosParam.bError;
			nErrId	:= ReadSercosParam.nErrId;
			ReadSercosParam(bExecute := FALSE);

			IF bError THEN
				(* error *)
				bIdnError		:= TRUE;
				nIdnErrId		:= nErrId;
				nIdnAccessId	:= nCRCIDN;
				bBusy			:= FALSE;
				eState 			:= eBkup_IDLE;
			ELSE
				(* read done, compare string *)
				bCheckOK 		:= (sCheckData.sString = sSavedCheckData.sString) AND (sCheckData.sString <> '');
				bBusy			:= FALSE;
				eState 			:= eBkup_IDLE;
			END_IF
		END_IF


	(*** read parameter list ***)
	eBkup_READ_IDNLIST_INI:
		(* first scan: initialization with rising edge on bExecute *)
		eState 			:= eBkup_READ_IDNLIST_ACT;

		IF bStdBackupList AND NOT(bCRCIDNTest) THEN
			nIDN		:= 192;
		ELSE
			nIDN		:= 17;
		END_IF

		ReadSercosParam(bExecute := FALSE);
		ReadSercosParam(
			sNetId 		:= sNetId,
			nIDN		:= nIDN,
			bExecute	:= TRUE,
			nMode		:= iVALUE,
			nPort		:= nPort,
			nAttrib		:= 0,
			cbLen		:= SIZEOF(arrList),
			dwDestAddr 	:= ADR(arrList),
			tTimeout	:= tTimeout
		);

	eBkup_READ_IDNLIST_ACT:
		(* following scans: wait for not busy *)
		ReadSercosParam(bExecute := FALSE);

		IF NOT(ReadSercosParam.bBusy) THEN
			(* not busy anymore *)
			bError	:= ReadSercosParam.bError;
			nErrId	:= ReadSercosParam.nErrId;
			ReadSercosParam(bExecute := FALSE);

			IF bError THEN
				(* error *)
				bBackupDone		:= FALSE;
				bRestoreDone	:= FALSE;
				bBackup_L	 	:= FALSE;
				bRestore_L	 	:= FALSE;
				bBusy			:= FALSE;
				eState 			:= eBkup_IDLE;
				bIdnError		:= TRUE;
				nIdnErrId		:= nErrId;
				nIdnAccessId	:= nIDN;
			ELSE
				(* done *)
				bEndOfList		:= FALSE;
				sListAttrib		:= ReadSercosParam.sAttrib;

				IF (sListAttrib.eType = eType_ID) AND (sListAttrib.eLength = eLEN_V2BYTE) THEN
					(* calculate number of list items *)
					nRetVal 		:= MEMCPY(ADR(iLastListItem), ADR(arrList[0]), SIZEOF(iLastListItem));
					iLastListItem 	:= iLastListItem / 2;
					iLastListItem 	:= LIMIT(0, iLastListItem, 32767);
					iActListItem	:= 0;
					nListArrIdx		:= 4;

					IF bCRCIDNTest THEN
						bCRCIDNTest  := FALSE;
						bCRCIDNExist := FALSE;

						FOR iIdx := 0 TO iLastListItem DO
							nRetVal := MEMCPY(ADR(iActListItem), ADR(arrList[nListArrIdx]), 2);
							nListArrIdx := nListArrIdx + 2;

							IF iActListItem = nCRCIDN THEN
								bCRCIDNExist := TRUE;
								EXIT;
							END_IF
						END_FOR

						IF bBackup_L OR bRestore_L THEN
							eState 	:= eBkup_READ_IDNLIST_INI;
						ELSE
							bBusy	:= FALSE;
							eState 	:= eBkup_IDLE;
						END_IF

					ELSE
						IF bBackup_L THEN
							eState 		:= eBkup_FILEOPEN;

							OpenBackupFile(
								sNetId 		:= sNetId,
								sPathName	:= sPathName,
								nMode		:= FOPEN_MODEWRITE OR FOPEN_MODEBINARY,
								ePath		:= ePath,
								bExecute	:= TRUE,
								tTimeout	:= tTimeout
							);

						ELSIF bRestore_L THEN
							eState 		:= eBkup_FILEOPEN;

							OpenBackupFile(
								sNetId 		:= sNetId,
								sPathName	:= sPathName,
								nMode		:= FOPEN_MODEREAD OR FOPEN_MODEBINARY,
								ePath		:= ePath,
								bExecute	:= TRUE,
								tTimeout	:= tTimeout
							);
						ELSE
							bBusy			:= FALSE;
							eState 			:= eBkup_IDLE;
						END_IF
					END_IF
				ELSE
					bBackupDone		:= FALSE;
					bRestoreDone	:= FALSE;
					bBackup_L	 	:= FALSE;
					bRestore_L	 	:= FALSE;
					bError			:= TRUE;
					nErrId			:= 16#1005;
					bBusy			:= FALSE;
					eState 			:= eBkup_IDLE;
				END_IF
			END_IF
		END_IF


	(*** backup current list ***)
	eBkup_FILEOPEN:
		OpenBackupFile(bExecute	:= FALSE);

		IF NOT(OpenBackupFile.bBusy) THEN
			bError	:= OpenBackupFile.bError;
			nErrId	:= OpenBackupFile.nErrId;
			OpenBackupFile(bExecute	:= FALSE);

			IF bError THEN
				(* error *)
				bBackupDone	:= FALSE;
				bRestoreDone:= FALSE;
				bBackup_L	:= FALSE;
				bRestore_L	:= FALSE;
				nFileErrId	:= nErrId;
				bBusy		:= FALSE;
				eState 		:= eBkup_IDLE;
				bFileOpen	:= FALSE;
				hFile		:= 0;
			ELSE
				bFileOpen	:= TRUE;
				hFile		:= OpenBackupFile.hFile;

				IF bBackup_L THEN
					(* preset header *)
					sFileHeader.nVersion 	 := nVersion;
					sFileHeader.nListType 	 := nIDN;
					sFileHeader.cbCommentLen := SIZEOF(sComment);
					nRetVal 				 := MEMCPY(ADR(sFileHeader.sComment), ADR(sComment), SIZEOF(sComment));

					WriteBackupFile(
						sNetId 		:= sNetId,
						hFile		:= hFile,
						pWriteBuff	:= ADR(sFileHeader),
						cbWriteLen	:= SIZEOF(sFileHeader),
						bExecute	:= TRUE,
						tTimeout	:= tTimeout
					);
					eState 	:= eBkup_BACKUP_WRITE_FILEHEADER;

				ELSIF bRestore_L THEN
					nRetVal := MEMSET(ADR(sFileHeader), 0, SIZEOF(sFileHeader));

					(* load header *)
					ReadBackupFile(
						sNetId 		:= sNetId,
						hFile		:= hFile,
						pReadBuff	:= ADR(sFileHeader),
						cbReadLen	:= SIZEOF(sFileHeader),
						bExecute	:= TRUE,
						tTimeout	:= tTimeout
					);
					eState 	:= eBkup_RESTORE_READ_FILEHEADER;
				END_IF
			END_IF
		END_IF


	(*** backup init ***)
	eBkup_BACKUP_WRITE_FILEHEADER:
		WriteBackupFile(bExecute := FALSE);

		IF NOT(WriteBackupFile.bBusy) THEN
			bError	:= WriteBackupFile.bError;
			nErrId	:= WriteBackupFile.nErrId;
			WriteBackupFile(bExecute := FALSE);

			IF bError THEN
				(* error *)
				bBackupDone	:= FALSE;
				bFileError	:= TRUE;
				nFileErrId	:= nErrId;
				bError		:= FALSE;
				nErrId		:= 0;
				eState 		:= eBkup_FILECLOSE;

				(* backup aborted *)
				CloseBackupFile(
					sNetId 		:= sNetId,
					hFile		:= hFile,
					bExecute	:= TRUE,
					tTimeout	:= tTimeout
				);

			ELSE
				cbSize 	:= WriteBackupFile.cbWrite;
				eState 	:= eBkup_BACKUP_PARAM_INI;
			END_IF
		END_IF

	(* backup current list *)
	eBkup_BACKUP_PARAM_INI:
		IF NOT(bEndOfList) THEN
			(* first scan: initialization with rising edge on bBackup *)
			bBackupDone			:= FALSE;

			(* get parameter *)
			IF (nListArrIdx >= 4) AND (nListArrIdx <= 65534) THEN
				eState 			:= eBkup_BACKUP_PARAM_ACT;
				nRetVal 		:= MEMCPY(ADR(nIDN), ADR(arrList[nListArrIdx]), SIZEOF(nIDN));
				nListArrIdx		:= nListArrIdx + SIZEOF(nIDN);

				ReadSercosParam(bExecute := FALSE);
				ReadSercosParam(
					sNetId 		:= sNetId,
					nIDN		:= nIDN,
					bExecute	:= TRUE,
					nMode		:= iVALUE,
					nPort		:= nPort,
					nAttrib		:= 0,
					cbLen		:= SIZEOF(arrData),
					dwDestAddr 	:= ADR(arrData),
					tTimeout	:= tTimeout
				);

			ELSE
				(* wrong index *)
				ReadSercosParam(bExecute := FALSE);
				iActListItem	:= 0;
				bBackupDone		:= FALSE;
				bIdnError		:= TRUE;
				bError			:= FALSE;
				nErrId			:= 0;
				eState 			:= eBkup_FILECLOSE;

				(* backup aborted *)
				CloseBackupFile(
					sNetId 		:= sNetId,
					hFile		:= hFile,
					bExecute	:= TRUE,
					tTimeout	:= tTimeout
				);
			END_IF
		ELSE
			(* backup completed *)
			ReadSercosParam(bExecute := FALSE);
			iActListItem	:= 0;
			eState 			:= eBkup_FILECLOSE;

			CloseBackupFile(
				sNetId 		:= sNetId,
				hFile		:= hFile,
				bExecute	:= TRUE,
				tTimeout	:= tTimeout
			);
		END_IF

	eBkup_BACKUP_PARAM_ACT:
		(* following scans: wait for not busy *)
		ReadSercosParam(bExecute := FALSE);

		IF NOT(ReadSercosParam.bBusy) THEN
			(* not busy anymore *)
			bError				:= ReadSercosParam.bError;
			nErrId				:= ReadSercosParam.nErrId;
			ReadSercosParam(bExecute := FALSE);

			IF bError THEN
				(* error *)
				bBackupDone		:= FALSE;
				bRestoreDone	:= FALSE;
				bIdnError		:= TRUE;
				nIdnErrId		:= nErrId;
				nIdnAccessId	:= nIDN;
				bError			:= FALSE;
				nErrId			:= 0;
				eState 			:= eBkup_FILECLOSE;

				(* backup aborted *)
				CloseBackupFile(
					sNetId 		:= sNetId,
					hFile		:= hFile,
					bExecute	:= TRUE,
					tTimeout	:= tTimeout
				);
			ELSE
				(* save data header *)
				sParamHeader.nIDN	:= ReadSercosParam.nIDN;
				sParamHeader.nAttrib:= ReadSercosParam.nAttribRd;
				sParamHeader.cbSize	:= UDINT_TO_UINT(ReadSercosParam.cbRead);

				(* update CRC16-CCITT and CheckSum *)
				IF nIDN <> nCRCIDN THEN
					wCRC16_CCITT	:= F_CRC16_CCITT(ADR(arrData), sParamHeader.cbSize, wCRC16_CCITT);
					wCheckSum		:= F_CheckSum16(ADR(arrData), sParamHeader.cbSize, wCheckSum);
				END_IF

				WriteBackupFile(
					sNetId 		:= sNetId,
					hFile		:= hFile,
					pWriteBuff	:= ADR(sParamHeader),
					cbWriteLen	:= SIZEOF(sParamHeader),
					bExecute	:= TRUE,
					tTimeout	:= tTimeout
				);

				eState 		:= eBkup_BACKUP_WRITE_HEADER;
			END_IF
		END_IF

	eBkup_BACKUP_WRITE_HEADER:
		WriteBackupFile(bExecute := FALSE);

		IF NOT(WriteBackupFile.bBusy) THEN
			bError	:= WriteBackupFile.bError;
			nErrId	:= WriteBackupFile.nErrId;
			WriteBackupFile(bExecute := FALSE);

			IF bError THEN
				(* error *)
				bBackupDone	:= FALSE;
				bFileError	:= TRUE;
				nFileErrId	:= nErrId;
				bError		:= FALSE;
				nErrId		:= 0;
				eState 		:= eBkup_FILECLOSE;

				(* backup aborted *)
				CloseBackupFile(
					sNetId 		:= sNetId,
					hFile		:= hFile,
					bExecute	:= TRUE,
					tTimeout	:= tTimeout
				);
			ELSE
				cbSize := WriteBackupFile.cbWrite;

				(* save data *)
				CASE sParamData.sAttrib.eLength OF
					eLEN_2BYTE,  eLEN_4BYTE,  eLEN_8BYTE,
					eLEN_V1BYTE, eLEN_V2BYTE, eLEN_V4BYTE, eLEN_V8BYTE:
						WriteBackupFile(
							sNetId 		:= sNetId,
							hFile		:= hFile,
							pWriteBuff	:= ADR(arrData),
							cbWriteLen	:= sParamHeader.cbSize,
							bExecute	:= TRUE,
							tTimeout	:= tTimeout
						);
				ELSE
					;
				END_CASE

				eState 		:= eBkup_BACKUP_WRITE_DATA;
			END_IF
		END_IF

	eBkup_BACKUP_WRITE_DATA:
		WriteBackupFile(bExecute := FALSE);

		IF NOT(WriteBackupFile.bBusy) THEN
			bError	:= WriteBackupFile.bError;
			nErrId	:= WriteBackupFile.nErrId;
			WriteBackupFile(bExecute := FALSE);

			IF bError THEN
				(* error *)
				bBackupDone	:= FALSE;
				bFileError	:= TRUE;
				nFileErrId	:= nErrId;
				bError		:= FALSE;
				nErrId		:= 0;
				eState 		:= eBkup_FILECLOSE;

				(* backup aborted *)
				CloseBackupFile(
					sNetId 		:= sNetId,
					hFile		:= hFile,
					bExecute	:= TRUE,
					tTimeout	:= tTimeout
				);
			ELSE
				cbSize 		:= WriteBackupFile.cbWrite;

				(* next item *)
				IF NOT(bEndOfList) THEN
					(* next item *)
					iActListItem		:= iActListItem + 1;

					(* backup next parameter *)
					eState 				:= eBkup_BACKUP_PARAM_INI;

					IF (iActListItem >= iLastListItem) THEN
						iActListItem	:= 0;
						bEndOfList		:= TRUE;

						(* backup completed *)
						ReadSercosParam(bExecute := FALSE);
						CloseBackupFile(
							sNetId 		:= sNetId,
							hFile		:= hFile,
							bExecute	:= TRUE,
							tTimeout	:= tTimeout
						);
						eState 		:= eBkup_FILECLOSE;
					END_IF
				ELSE
					(* backup completed *)
					CloseBackupFile(
						sNetId 		:= sNetId,
						hFile		:= hFile,
						bExecute	:= TRUE,
						tTimeout	:= tTimeout
					);
					ReadSercosParam(bExecute := FALSE);
					eState 		:= eBkup_FILECLOSE;
				END_IF
			END_IF
		END_IF


	(*** restore init ***)
	eBkup_RESTORE_READ_FILEHEADER:
		ReadBackupFile(bExecute := FALSE);

		IF NOT(ReadBackupFile.bBusy) THEN
			bError	:= ReadBackupFile.bError;
			nErrId	:= ReadBackupFile.nErrId;
			ReadBackupFile(bExecute := FALSE);

			IF bError THEN
				(* error *)
				bRestoreDone:= FALSE;
				bFileError	:= TRUE;
				nFileErrId	:= nErrId;
				bError		:= FALSE;
				nErrId		:= 0;
				eState 		:= eBkup_FILECLOSE;

				(* backup aborted *)
				CloseBackupFile(
					sNetId 		:= sNetId,
					hFile		:= hFile,
					bExecute	:= TRUE,
					tTimeout	:= tTimeout
				);
			ELSE
				cbSize 			:= ReadBackupFile.cbRead;
				sComment		:= sFileHeader.sComment;

				IF sFileHeader.nListType = 192 THEN
					bWrongListType	:= FALSE;

					ReadBackupFile(
						sNetId 		:= sNetId,
						hFile		:= hFile,
						pReadBuff	:= ADR(sParamHeader),
						cbReadLen	:= SIZEOF(sParamHeader),
						bExecute	:= TRUE,
						tTimeout	:= tTimeout
					);
					eState 			:= eBkup_RESTORE_READ_HEADER;
				ELSE
					bWrongListType	:= TRUE;

					(* backup completed *)
					CloseBackupFile(
						sNetId 		:= sNetId,
						hFile		:= hFile,
						bExecute	:= TRUE,
						tTimeout	:= tTimeout
					);
					eState 		:= eBkup_FILECLOSE;
				END_IF
			END_IF
		END_IF

	eBkup_RESTORE_READ_HEADER:
		ReadBackupFile(bExecute := FALSE);

		IF NOT(ReadBackupFile.bBusy) THEN
			bError	:= ReadBackupFile.bError;
			nErrId	:= ReadBackupFile.nErrId;
			ReadBackupFile(bExecute := FALSE);

			IF bError THEN
				(* error *)
				bRestoreDone:= FALSE;
				bFileError	:= TRUE;
				nFileErrId	:= nErrId;
				bError		:= FALSE;
				nErrId		:= 0;
				eState 		:= eBkup_FILECLOSE;

				(* backup aborted *)
				CloseBackupFile(
					sNetId 		:= sNetId,
					hFile		:= hFile,
					bExecute	:= TRUE,
					tTimeout	:= tTimeout
				);
			ELSE
				cbSize := sParamHeader.cbSize;

				IF (ReadBackupFile.cbRead <> 0) THEN
					nRetVal		:= MEMSET(ADR(arrData[0]), 0, SIZEOF(arrData));

					ReadBackupFile(
						sNetId 		:= sNetId,
						hFile		:= hFile,
						pReadBuff	:= ADR(arrData),
						cbReadLen	:= sParamHeader.cbSize,
						bExecute	:= TRUE,
						tTimeout	:= tTimeout
					);
					eState 			:= eBkup_RESTORE_READ_DATA;
				ELSE
					(* backup completed *)
					CloseBackupFile(
						sNetId 		:= sNetId,
						hFile		:= hFile,
						bExecute	:= TRUE,
						tTimeout	:= tTimeout
					);
					eState 		:= eBkup_FILECLOSE;
				END_IF
			END_IF
		END_IF

	eBkup_RESTORE_READ_DATA:
		ReadBackupFile(bExecute := FALSE);

		IF NOT(ReadBackupFile.bBusy) THEN
			bError		:= ReadBackupFile.bError;
			nErrId		:= ReadBackupFile.nErrId;
			ReadBackupFile(bExecute := FALSE);

			IF bError THEN
				(* error *)
				bRestoreDone:= FALSE;
				bFileError	:= TRUE;
				nFileErrId	:= nErrId;
				bError		:= FALSE;
				nErrId		:= 0;
				eState 		:= eBkup_FILECLOSE;

				(* backup aborted *)
				CloseBackupFile(
					sNetId 		:= sNetId,
					hFile		:= hFile,
					bExecute	:= TRUE,
					tTimeout	:= tTimeout
				);
			ELSE
				IF ReadBackupFile.bEOF THEN
					bEndOfList	:= TRUE;
				END_IF

				cbSize 	:= ReadBackupFile.cbRead;
				eState 	:= eBkup_RESTORE_PARAM_INI;
			END_IF
		END_IF

	(* restore current list item *)
	eBkup_RESTORE_PARAM_INI:
		(* first scan: initialization with rising edge on bBackup *)
		bRestoreDone	:= FALSE;
		eState 			:= eBkup_RESTORE_PARAM_ACT;
		nIDN			:= sParamHeader.nIDN;

		sParamData.nAttrib					:= sParamHeader.nAttrib;

		(* split attribute *)
		sParamData.sAttrib.nFactor			:= DWORD_TO_UINT(sParamHeader.nAttrib AND 16#0000FFFF); 			(* bits  0..15 *)
		sParamData.sAttrib.eLength			:= DWORD_TO_INT(SHR(sParamHeader.nAttrib, 16) AND 16#00000007);		(* bits 16..18 *)
		sParamData.sAttrib.bCommand			:= DWORD_TO_BOOL(SHR(sParamHeader.nAttrib, 19) AND 16#00000001);	(* bit  19     *)
		sParamData.sAttrib.eType			:= DWORD_TO_INT(SHR(sParamHeader.nAttrib, 20) AND 16#00000007);		(* bits 20..22 *)
		sParamData.sAttrib.bReserved1		:= DWORD_TO_BOOL(SHR(sParamHeader.nAttrib, 23) AND 16#00000001);	(* bit  23     *)
		sParamData.sAttrib.nComma			:= DWORD_TO_USINT(SHR(sParamHeader.nAttrib, 24) AND 16#0000000F);	(* bits 24..27 *)
		sParamData.sAttrib.bWriteProtCP2	:= DWORD_TO_BOOL(SHR(sParamHeader.nAttrib, 28) AND 16#00000001);	(* bit  28     *)
		sParamData.sAttrib.bWriteProtCP3	:= DWORD_TO_BOOL(SHR(sParamHeader.nAttrib, 29) AND 16#00000001);	(* bit  29     *)
		sParamData.sAttrib.bWriteProtCP4	:= DWORD_TO_BOOL(SHR(sParamHeader.nAttrib, 30) AND 16#00000001);	(* bit  30     *)
		sParamData.sAttrib.bReserved2		:= DWORD_TO_BOOL(SHR(sParamHeader.nAttrib, 31) AND 16#00000001);	(* bit  31     *)

		CASE sParamData.sAttrib.eLength OF
			eLEN_2BYTE:
				cbLen	:= 2;

			eLEN_4BYTE:
				cbLen	:= 4;

			eLEN_8BYTE:
				cbLen	:= 8;

			eLEN_V1BYTE, eLEN_V2BYTE, eLEN_V4BYTE, eLEN_V8BYTE:
				nRetVal := MEMCPY(ADR(cbLen), ADR(arrData), 2);
				cbLen	:= cbLen + 4; (* act len & max len *)
		ELSE
			cbLen	:= 0;
		END_CASE

		WriteSercosParam(bExecute := FALSE);
		WriteSercosParam(
			sNetId 		:= sNetId,
			nIDN		:= nIDN,
			bExecute	:= TRUE,
			nPort		:= nPort,
			nAttrib		:= sParamData.nAttrib,
			cbLen		:= cbLen,
			dwSrcAddr	:= ADR(arrData),
			tTimeout	:= tTimeout
		);

	eBkup_RESTORE_PARAM_ACT:
		(* following scans: wait for not busy *)
		WriteSercosParam(bExecute := TRUE);

		IF NOT(WriteSercosParam.bBusy) THEN
			(* not busy anymore *)
			bError				:= WriteSercosParam.bError;
			nErrId				:= WriteSercosParam.nErrId;
			WriteSercosParam(bExecute := FALSE);

			IF bError THEN
				(* error *)
				bBackupDone		:= FALSE;
				bRestoreDone	:= FALSE;
				bIdnError		:= TRUE;
				nIdnErrId		:= nErrId;
				nIdnAccessId	:= nIDN;
				bError			:= FALSE;
				nErrId			:= 0;
				eState 			:= eBkup_FILECLOSE;

				(* backup aborted *)
				CloseBackupFile(
					sNetId 		:= sNetId,
					hFile		:= hFile,
					bExecute	:= TRUE,
					tTimeout	:= tTimeout
				);

			ELSE
				(* update CRC16-CCITT and CheckSum *)
				IF nIDN <> nCRCIDN THEN
					wCRC16_CCITT	:= F_CRC16_CCITT(ADR(arrData), cbLen, wCRC16_CCITT);
					wCheckSum		:= F_CheckSum16(ADR(arrData), cbLen, wCheckSum);
				END_IF

				(* next parameter *)
				iActListItem	:= iActListItem + 1;

				IF NOT(bEndOfList) THEN
					ReadBackupFile(
						sNetId 		:= sNetId,
						hFile		:= hFile,
						pReadBuff	:= ADR(sParamHeader),
						cbReadLen	:= SIZEOF(sParamHeader),
						bExecute	:= TRUE,
						tTimeout	:= tTimeout
					);
					eState 			:= eBkup_RESTORE_READ_HEADER;
				ELSE
					(* backup completed *)
					CloseBackupFile(
						sNetId 		:= sNetId,
						hFile		:= hFile,
						bExecute	:= TRUE,
						tTimeout	:= tTimeout
					);
					WriteSercosParam(bExecute := FALSE);
					eState 		:= eBkup_FILECLOSE;
				END_IF
			END_IF
		END_IF

	(*** done or aborted  ***)
	eBkup_FILECLOSE:
		CloseBackupFile(bExecute := FALSE);

		IF NOT(CloseBackupFile.bBusy) THEN
			bError	:= CloseBackupFile.bError;
			nErrId	:= CloseBackupFile.nErrId;
			CloseBackupFile(bExecute := FALSE);

			IF bError THEN
				(* error *)
				bBackupDone	:= FALSE;
				bRestoreDone:= FALSE;
				bBackup_L	:= FALSE;
				bRestore_L	:= FALSE;
				bBusy		:= FALSE;
				eState 		:= eBkup_IDLE;
			ELSE
				bFileOpen	:= FALSE;
				hFile		:= 0;

				IF bUpdateCRC AND bCRCEnable THEN
					IF NOT(bFileError OR bIdnError) THEN
						sCheckData.sString := 'CRC= ';
						sCheckData.sString := CONCAT(sCheckData.sString, WORD_TO_STRING(wCRC16_CCITT));
						sCheckData.sString := CONCAT(sCheckData.sString, ', ChkSum= ');
						sCheckData.sString := CONCAT(sCheckData.sString, WORD_TO_STRING(wCheckSum));

						IF bBackup_L OR (bRestore_L AND NOT(bWrongListType)) THEN
							ReadSercosParam(bExecute := FALSE);
							ReadSercosParam(
								sNetId 		:= sNetId,
								nIDN		:= nCRCIDN,
								bExecute	:= TRUE,
								nMode		:= iVALUE,
								nPort		:= nPort,
								nAttrib		:= 0,
								cbLen		:= 4,
								dwDestAddr 	:= ADR(sCheckData),
								tTimeout	:= tTimeout
							);

							eState		 := eBkup_UPDT_CRC_INI;
						ELSE
							IF bWrongListType THEN
								bBackupDone := FALSE;
								bRestoreDone:= FALSE;
								bBackup_L	:= FALSE;
								bRestore_L	:= FALSE;
								bError		:= TRUE;
								nErrId		:= 16#1006;	(* backup list was NOT IDN 192 *)
								bBusy		:= FALSE;
								eState 		:= eBkup_IDLE;
							END_IF
						END_IF
					END_IF
				ELSE
					(* done, no CRC and check sum *)
					IF bBackup_L THEN
						bBackup_L	:= FALSE;
						bBackupDone	:= TRUE;
					ELSIF bRestore_L THEN
						bRestore_L	:= FALSE;
						bRestoreDone:= TRUE;
					END_IF

					bBusy		:= FALSE;
					eState 		:= eBkup_IDLE;
				END_IF

				IF bFileError THEN
					bError		 := TRUE;
					nErrId		 := nFileErrId;
					bUpdateCRC	 := FALSE;
					bRestoreDone := FALSE;
					bBackupDone	 := FALSE;
					bBackup_L	 := FALSE;
					bRestore_L	 := FALSE;
					bBusy		 := FALSE;
					eState 		 := eBkup_IDLE;
				ELSIF bIdnError THEN
					bError		 := TRUE;
					nErrId		 := nIdnErrId;
					bUpdateCRC	 := FALSE;
					bRestoreDone := FALSE;
					bBackupDone	 := FALSE;
					bBackup_L	 := FALSE;
					bRestore_L	 := FALSE;
					bBusy		 := FALSE;
					eState 		 := eBkup_IDLE;
				END_IF
			END_IF
		END_IF

	eBkup_UPDT_CRC_INI:
		ReadSercosParam(bExecute := FALSE);

		IF NOT(ReadSercosParam.bBusy) THEN
			(* not busy anymore *)
			bError	:= ReadSercosParam.bError;
			nErrId	:= ReadSercosParam.nErrId;
			ReadSercosParam(bExecute := FALSE);

			IF bError THEN
				(* error *)
				bRestoreDone 	:= FALSE;
				bBackupDone	 	:= FALSE;
				bBackup_L	 	:= FALSE;
				bRestore_L	 	:= FALSE;
				bUpdateCRC	 	:= FALSE;
				bIdnError		:= TRUE;
				nIdnErrId		:= nErrId;
				nIdnAccessId	:= nCRCIDN;
				bBusy			:= FALSE;
				eState 			:= eBkup_IDLE;
			ELSE
				sCheckData.iActSize:= LEN(sCheckData.sString);
				sParamData.nAttrib	:= ReadSercosParam.nAttribRd;

				WriteSercosParam(bExecute := FALSE);
				WriteSercosParam(
					sNetId 		:= sNetId,
					nIDN		:= nCRCIDN,
					bExecute	:= TRUE,
					nPort		:= nPort,
					nAttrib		:= sParamData.nAttrib,
					cbLen		:= sCheckData.iActSize + 4,
					dwSrcAddr	:= ADR(sCheckData),
					tTimeout	:= tTimeout
				);

				eState		 := eBkup_UPDT_CRC_ACT;
			END_IF
		END_IF

	eBkup_UPDT_CRC_ACT:
		(* wait for CRC updated *)
		WriteSercosParam(bExecute := FALSE);

		IF NOT(WriteSercosParam.bBusy) THEN
			(* not busy anymore *)
			bError				:= WriteSercosParam.bError;
			nErrId				:= WriteSercosParam.nErrId;
			WriteSercosParam(bExecute := FALSE);
			bUpdateCRC	 		:= FALSE;

			IF bError THEN
				(* error *)
				bRestoreDone 	:= FALSE;
				bBackupDone	 	:= FALSE;
				bBackup_L	 	:= FALSE;
				bRestore_L	 	:= FALSE;
				bBusy			:= FALSE;
				eState 			:= eBkup_IDLE;
				bIdnError		:= TRUE;
				nIdnErrId		:= nErrId;
				nIdnAccessId	:= nIDN;
				bError			:= FALSE;
				nErrId			:= 0;

			ELSE
				(* done *)
				IF bBackup_L THEN
					bBackup_L	:= FALSE;
					bBackupDone	:= TRUE;
				ELSIF bRestore_L THEN
					bRestore_L	:= FALSE;
					bRestoreDone:= TRUE;
				END_IF

				bBusy			:= FALSE;
				eState 			:= eBkup_IDLE;

				(* update CRC16-CCITT and CheckSum *)
				wSavedCRC16_CCITT := wCRC16_CCITT;
				wSavedCheckSum	  := wCheckSum;
				sSavedCheckData	  := sCheckData;
			END_IF
		END_IF

ELSE
	(* undefined state *)
	bRestoreDone:= FALSE;
	bBackupDone	:= FALSE;
	bBackup_L	:= FALSE;
	bRestore_L	:= FALSE;
	bBusy		:= FALSE;
	bError		:= TRUE;
	bUpdateCRC	:= FALSE;
	eState 		:= eBkup_IDLE;
END_CASE

(* clear current data for edge detection *)
bBackup_I 	:= bBackup_I AND bBackup;
bRestore_I 	:= bRestore_I AND bRestore;
bCheck_I 	:= bCheck_I AND bCheck;
END_FUNCTION_BLOCK

(* POU IOF_SER_IDN_Read, ST *)
FUNCTION_BLOCK IOF_SER_IDN_Read
VAR_INPUT
	sNetId 				: T_AmsNetId;	(* ams net id *)
	nIDN				: UINT;			(* S: 0******* ********, P: 1******* ******** *)
	bExecute			: BOOL;			(* starts read with rising edge *)
	nPort				: UINT;			(* sercos axis ads port number *)
	nMode				: DINT;			(* read: 0= Value, 2= Name, 3= Attribute, 4= Unit, 5= Minimum, 6= Maximum *)
	nAttrib				: DWORD;		(* parameter attribute if known, otherwise 0 *)
	cbLen				: UDINT;		(* max lenght of data buffer *)
	dwDestAddr 		: DWORD;		(* address of data buffer *)
	tTimeout			: TIME := DEFAULT_ADS_TIMEOUT;	(* timeout for complete parameter access (e.g. incl. attribute) *)
END_VAR
VAR_OUTPUT
	cbRead				: UDINT;
	nAttribRd			: DWORD;
	sAttrib				: ST_SercosParamAttrib;
	bBusy 				: BOOL;
	bError				: BOOL;
	nErrId 				: UDINT;
(*	Function block specific error codes:
	16#1003 =  Wrong parameter mode
	16#1004 = Data parameter wrong value size
*)
END_VAR
VAR
	ReadBlock 			: ADSREAD;
	iState				: INT;
	iRepeats			: INT;
	nRetVal				: UDINT;
	dwDestAddr_I		: DWORD;
	bExecute_I			: BOOL;
	nMode_I				: DINT;
	Timeout				: TON := (PT := T#100ms);
END_VAR
VAR CONSTANT
	iVALUE				: DINT := 0;		(* Parameter Value *)
	iFCNSTATE			: DINT := 1;		(* Function State *)
	iNAME				: DINT := 2;		(* Parameter Name *)
	iATTRIB				: DINT := 3;		(* Parameter Attribute *)
	iUNIT				: DINT := 4;		(* Parameter Unit *)
	iMIN				: DINT := 5;		(* Parameter Minimum *)
	iMAX				: DINT := 6;		(* Parameter Maximum *)
END_VAR
(* state machine *)
CASE iState OF
0:	(* wait for rising edge *)
	IF bExecute AND NOT(bExecute_I) THEN
		bBusy    := TRUE;
		bError 	 := FALSE;
		nErrId 	 := 0;
		iRepeats := 0;
		nMode_I  := nMode;

		(* clear data *)
		cbRead	 := 0;
		nRetVal  := MEMSET(dwDestAddr, 0, cbLen);

		Timeout(IN := FALSE);
		ReadBlock(READ := FALSE);

		IF (nAttrib <> 0) THEN
			sAttrib.nFactor			:= DWORD_TO_UINT(nAttrib          AND 16#0000FFFF); (* bits  0..15 *)
			sAttrib.eLength			:= DWORD_TO_INT(SHR(nAttrib,  16) AND 16#00000007);	(* bits 16..18 *)
			sAttrib.bCommand		:= DWORD_TO_BOOL(SHR(nAttrib, 19) AND 16#00000001);	(* bit  19     *)
			sAttrib.eType			:= DWORD_TO_INT(SHR(nAttrib,  20) AND 16#00000007);	(* bits 20..22 *)
			sAttrib.bReserved1		:= DWORD_TO_BOOL(SHR(nAttrib, 23) AND 16#00000001);	(* bit  23     *)
			sAttrib.nComma			:= DWORD_TO_USINT(SHR(nAttrib,24) AND 16#0000000F); (* bits 24..27 *)
			sAttrib.bWriteProtCP2	:= DWORD_TO_BOOL(SHR(nAttrib, 28) AND 16#00000001);	(* bit  28     *)
			sAttrib.bWriteProtCP3	:= DWORD_TO_BOOL(SHR(nAttrib, 29) AND 16#00000001);	(* bit  29     *)
			sAttrib.bWriteProtCP4	:= DWORD_TO_BOOL(SHR(nAttrib, 30) AND 16#00000001);	(* bit  30     *)
			sAttrib.bReserved2		:= DWORD_TO_BOOL(SHR(nAttrib, 31) AND 16#00000001);	(* bit  31     *)
		END_IF

		IF (nAttrib = 0) OR (sAttrib.eLength = 0) OR (nMode = iATTRIB) THEN
			(* read attrib first, read other data afterwards *)
			iState 		:= 1;
			nAttribRd	:= 0;
			nRetVal 	:= MEMSET(ADR(sAttrib), 0, SIZEOF(sAttrib));
		ELSE
			(* use known attrib, read other data immediatelly *)
			nAttribRd	:= nAttrib;

			CASE nMode_I OF
			iVALUE:
				iState := 3;

			iNAME:
				iState := 5;

			iUNIT:
				iState := 7;

			iMIN:
				iState := 9;

			iMAX:
				iState := 11;

			iFCNSTATE:
				iState := 13;

			ELSE
				(* error *)
				bError := TRUE;
				nErrId := 16#1003; (*  Wrong parameter mode *)
				bBusy  := FALSE;
				iState := 0;
			END_CASE
		END_IF
	END_IF

1:	(* read attrib init *)
	iState 	 	:= 2;
	nAttribRd	:= 0;
	cbRead 		:= SIZEOF(nAttribRd);
	dwDestAddr_I:= ADR(nAttribRd);

	ReadBlock(
		NETID 		:= sNetId,
		PORT 		:= nPort,
		IDXGRP 		:= nIDN,
		IDXOFFS 	:= iATTRIB,
		LEN 		:= cbRead,
		DESTADDR 	:= dwDestAddr_I,
		READ 		:= TRUE,
		TMOUT 		:= tTimeout
	);
	Timeout(IN := FALSE);

2:	(* read attrib act *)
	ReadBlock(READ := FALSE);

	IF NOT(ReadBlock.BUSY) THEN
		ReadBlock(READ := FALSE);

		IF NOT(ReadBlock.ERR) THEN
			(* split attribute *)
			sAttrib.nFactor			:= DWORD_TO_UINT(nAttribRd          AND 16#0000FFFF); 	(* bits  0..15 *)
			sAttrib.eLength			:= DWORD_TO_INT(SHR(nAttribRd,  16) AND 16#00000007);	(* bits 16..18 *)
			sAttrib.bCommand		:= DWORD_TO_BOOL(SHR(nAttribRd, 19) AND 16#00000001);	(* bit  19     *)
			sAttrib.eType			:= DWORD_TO_INT(SHR(nAttribRD,  20) AND 16#00000007);	(* bits 20..22 *)
			sAttrib.bReserved1		:= DWORD_TO_BOOL(SHR(nAttribRd, 23) AND 16#00000001);	(* bit  23     *)
			sAttrib.nComma			:= DWORD_TO_USINT(SHR(nAttribRd,24) AND 16#0000000F);	(* bits 24..27 *)
			sAttrib.bWriteProtCP2	:= DWORD_TO_BOOL(SHR(nAttribRd, 28) AND 16#00000001);	(* bit  28     *)
			sAttrib.bWriteProtCP3	:= DWORD_TO_BOOL(SHR(nAttribRd, 29) AND 16#00000001);	(* bit  29     *)
			sAttrib.bWriteProtCP4	:= DWORD_TO_BOOL(SHR(nAttribRd, 30) AND 16#00000001);	(* bit  30     *)
			sAttrib.bReserved2		:= DWORD_TO_BOOL(SHR(nAttribRd, 31) AND 16#00000001);	(* bit  31     *)

			CASE nMode_I OF
			iATTRIB:
				nRetVal := MEMCPY(dwDestAddr, ADR(nAttribRd), MIN(SIZEOF(nAttribRd), cbLen));
				cbRead	:= nRetVal;
				bBusy   := FALSE;
				iState  := 0;

			iVALUE:
				iState := 3;

			iNAME:
				iState := 5;

			iUNIT:
				iState := 7;

			iMIN:
				iState := 9;

			iMAX:
				iState := 11;

			iFCNSTATE:
				iState := 13;

			ELSE
				(* error *)
				bError := TRUE;
				nErrId := 16#1003; (*  Wrong parameter mode *)
				bBusy  := FALSE;
				iState := 0;
			END_CASE

			ReadBlock(READ := FALSE);
			iRepeats := 0;
		ELSE
			(* Timeout error *)
			IF (ReadBlock.ErrId = 16#745) AND (iRepeats <= 3) THEN
				Timeout(IN := TRUE);

				IF Timeout.Q THEN
					Timeout(IN := FALSE);
					(* retry request 3 times after timeout of 10 ms *)

					ReadBlock(READ := FALSE); (* create rising edge *)
					iRepeats := iRepeats + 1;
					iState 	 := 1;
				END_IF

			(* report other errors immeditelly *)
			ELSE
				bError 		:= ReadBlock.ERR;
				nErrId  	:= ReadBlock.ERRID;
				bBusy     	:= FALSE;
				iState 		:= 0;

				Timeout(IN := FALSE);
				ReadBlock( READ := FALSE );
			END_IF
		END_IF
	END_IF

3:	(* read value init *)
	iState 		 := 4;
	dwDestAddr_I := dwDestAddr;

	CASE sAttrib.eLength OF
		eLEN_2BYTE:
			cbRead 	   := 2;

		eLEN_4BYTE:
			cbRead 	 := 4;

		eLEN_8BYTE:
			cbRead 	 := 8;

		eLEN_V1BYTE, eLEN_V2BYTE, eLEN_V4BYTE, eLEN_V8BYTE:
			cbRead 	 := cbLen;

	ELSE
		bError	:= TRUE;
		nErrId	:= 16#1004; (* Data parameter wrong value size *)
		bBusy	:= FALSE;
		iState  := 0;
	END_CASE

	cbRead 	 	:= LIMIT(0, cbRead, cbLen);

	IF NOT(bError) THEN
		ReadBlock(
			NETID 		:= sNetId,
			PORT 		:= nPort,
			IDXGRP 		:= nIDN,
			IDXOFFS 	:= iVALUE,
			LEN 		:= cbRead,
			DESTADDR 	:= dwDestAddr_I,
			READ 		:= TRUE,
			TMOUT 		:= tTimeout
		);
		Timeout(IN := FALSE);
	END_IF

4:	(* read value act *)
	ReadBlock(READ := FALSE);

	IF NOT(ReadBlock.BUSY) THEN
		ReadBlock(READ := FALSE);

		IF NOT(ReadBlock.ERR) THEN
			CASE sAttrib.eLength OF
				eLEN_V1BYTE, eLEN_V2BYTE, eLEN_V4BYTE, eLEN_V8BYTE:
					cbRead	:= 0;
					nRetVal := MEMCPY(ADR(cbRead), dwDestAddr_I, 2);
					cbRead	:= cbRead + 4; (* act len & max len *)

				eLEN_2BYTE, eLEN_4BYTE, eLEN_8BYTE:
					;
			ELSE
				bError	:= TRUE;
				nErrId	:= 16#1004; (* Data parameter wrong value size *)
				bBusy	:= FALSE;
				iState	:= 0;
			END_CASE

			IF NOT(bError) THEN
				(* done *)
				iState	:= 0;
				bBusy	:= FALSE;
			END_IF

			iRepeats 	:= 0;
			ReadBlock(READ := FALSE);
		ELSE
			(* Timeout error *)
			IF (ReadBlock.ErrId = 16#745) AND (iRepeats <= 3) THEN
				Timeout(IN := TRUE);

				IF Timeout.Q THEN
					Timeout(IN := FALSE);
					(* retry request 3 times after timeout of 10 ms *)

					ReadBlock(READ := FALSE); (* create rising edge *)
					iRepeats := iRepeats + 1;
					iState	 := 3;
				END_IF

			(* report other errors immeditelly *)
			ELSE
				bError 	:= ReadBlock.ERR;
				nErrId  := ReadBlock.ERRID;
				bBusy   := FALSE;
				iState	:= 0;

				Timeout(IN := FALSE);
				ReadBlock(READ := FALSE);
			END_IF
		END_IF
	END_IF

5:	(* read name init *)
	iState	 	 := 6;
	cbRead		 := cbLen;
	dwDestAddr_I := dwDestAddr;

	ReadBlock(
		NETID 		:= sNetId,
		PORT 		:= nPort,
		IDXGRP 		:= nIDN,
		IDXOFFS 	:= iNAME,
		LEN 		:= cbRead,
		DESTADDR 	:= dwDestAddr_I,
		READ 		:= TRUE,
		TMOUT 		:= tTimeout
	);
	Timeout(IN := FALSE);

6:	(* read name act *)
	ReadBlock(READ := FALSE);

	IF NOT(ReadBlock.BUSY) THEN
		ReadBlock(READ := FALSE);

		IF NOT(ReadBlock.ERR) THEN
			(* done *)
			cbRead	:= 0;
			nRetVal := MEMCPY(ADR(cbRead), dwDestAddr_I, 2);
			cbRead	:= cbRead + 4;
			iState  := 0;
			bBusy   := FALSE;

			ReadBlock(READ := FALSE);
			iRepeats := 0;
		ELSE
			(* Timeout error *)
			IF (ReadBlock.ErrId = 16#745) AND (iRepeats <= 3) THEN
				Timeout(IN := TRUE);

				IF Timeout.Q THEN
					Timeout(IN := FALSE);
					(* retry request 3 times after timeout of 10 ms *)

					ReadBlock(READ := FALSE); (* create rising edge *)
					iRepeats := iRepeats + 1;
					iState	 := 5;
				END_IF

			(* report other errors immeditelly *)
			ELSE
				bError 	:= ReadBlock.ERR;
				nErrId  := ReadBlock.ERRID;
				bBusy   := FALSE;
				iState	:= 0;

				Timeout(IN := FALSE);
				ReadBlock(READ := FALSE);
			END_IF
		END_IF
	END_IF

7:	(* read unit init *)
	iState	 	 := 8;
	cbRead		 := cbLen;
	dwDestAddr_I := dwDestAddr;

	ReadBlock(
		NETID 		:= sNetId,
		PORT 		:= nPort,
		IDXGRP 		:= nIDN,
		IDXOFFS 	:= iUNIT,
		LEN 		:= cbRead,
		DESTADDR 	:= dwDestAddr_I,
		READ 		:= TRUE,
		TMOUT 		:= tTimeout
	);
	Timeout(IN := FALSE);

8:	(* read unit act *)
	ReadBlock(READ := FALSE);

	IF NOT(ReadBlock.BUSY) THEN
		ReadBlock(READ := FALSE);

		IF NOT(ReadBlock.ERR) THEN
			(* done *)
			cbRead	:= 0;
			nRetVal := MEMCPY(ADR(cbRead), dwDestAddr_I, 2);
			cbRead	:= cbRead + 4;
			iState  := 0;
			bBusy   := FALSE;

			ReadBlock(READ := FALSE);
			iRepeats := 0;
		ELSE
			(* Timeout error *)
			IF (ReadBlock.ErrId = 16#745) AND (iRepeats <= 3) THEN
				Timeout(IN := TRUE);

				IF Timeout.Q THEN
					Timeout(IN := FALSE);
					(* retry request 3 times after timeout of 10 ms *)

					ReadBlock(READ := FALSE); (* create rising edge *)
					iRepeats := iRepeats + 1;
					iState	 := 7;
				END_IF

			(* report other errors immeditelly *)
			ELSE
				bError 	:= ReadBlock.ERR;
				nErrId  := ReadBlock.ERRID;
				bBusy   := FALSE;
				iState	:= 0;

				Timeout(IN := FALSE);
				ReadBlock(READ := FALSE);
			END_IF
		END_IF
	END_IF

9:	(* read min init *)
	iState	 	 := 10;
	dwDestAddr_I := dwDestAddr;

	CASE sAttrib.eLength OF
		eLEN_2BYTE:
			cbRead	 := 2;

		eLEN_4BYTE:
			cbRead	 := 4;

		eLEN_8BYTE:
			cbRead 	 := 8;

	ELSE
		cbRead 	 := 0;
		bError	 := TRUE;
		nErrId	:= 16#1004; (* Data parameter wrong value size *)
		bBusy	 := FALSE;
		iState 	 := 0;
	END_CASE

	cbRead 	 	:= LIMIT(0, cbRead, cbLen);

